gfCNCPoint4[18037] = {X 357.4015, Y 26.8104, Z -5.5000, A 0.000, B 0.000, C 0.000 }
gfCNCPoint4[18038] = {X 357.5143, Y 25.0808, Z -5.5000, A 0.000, B 0.000, C 0.000 }
gfCNCPoint4[18039] = {X 357.4620, Y 23.3484, Z -5.5000, A 0.000, B 0.000, C 0.000 }
gfCNCPoint4[18040] = {X 357.2450, Y 21.6288, Z -5.5000, A 0.000, B 0.000, C 0.000 }
gfCNCPoint4[18041] = {X 356.8838, Y 20.0827, Z -5.5000, A 0.000, B 0.000, C 0.000 }
gfCNCPoint4[18042] = {X 356.3231, Y 18.5973, Z -5.5000, A 0.000, B 0.000, C 0.000 }
gfCNCPoint4[18043] = {X 355.5723, Y 17.1983, Z -5.5000, A 0.000, B 0.000, C 0.000 }
gfCNCPoint4[18044] = {X 354.6445, Y 15.9099, Z -5.5000, A 0.000, B 0.000, C 0.000 }
gfCNCPoint4[18045] = {X 353.7511, Y 14.9589, Z -5.5000, A 0.000, B 0.000, C 0.000 }
gfCNCPoint4[18046] = {X 352.7344, Y 14.1410, Z -5.5000, A 0.000, B 0.000, C 0.000 }
gfCNCPoint4[18047] = {X 351.6142, Y 13.4719, Z -5.5000, A 0.000, B 0.000, C 0.000 }
gfCNCPoint4[18048] = {X 350.4121, Y 12.9645, Z -5.5000, A 0.000, B 0.000, C 0.000 }
gfCNCPoint4[18049] = {X 349.1512, Y 12.6287, Z -5.5000, A 0.000, B 0.000, C 0.000 }
gfCNCPoint4[18050] = {X 347.5974, Y 12.4216, Z -5.5000, A 0.000, B 0.000, C 0.000 }
gfCNCPoint4[18051] = {X 346.0300, Y 12.3943, Z -5.5000, A 0.000, B 0.000, C 0.000 }
gfCNCPoint4[18052] = {X 344.4699, Y 12.5474, Z -5.5000, A 0.000, B 0.000, C 0.000 }
gfCNCPoint4[18053] = {X 342.9377, Y 12.8786, Z -5.5000, A 0.000, B 0.000, C 0.000 }
gfCNCPoint4[18054] = {X 341.4538, Y 13.3837, Z -5.5000, A 0.000, B 0.000, C 0.000 }
gfCNCPoint4[18055] = {X 340.0376, Y 14.0559, Z -5.5000, A 0.000, B 0.000, C 0.000 }
gfCNCPoint4[18056] = {X 338.7081, Y 14.8864, Z -5.5000, A 0.000, B 0.000, C 0.000 }
gfCNCPoint4[18057] = {X 338.6941, Y 15.7112, Z -5.5000, A 0.000, B 0.000, C 0.000 }
gfCNCPoint4[18058] = {X 338.5145, Y 16.5162, Z -5.5000, A 0.000, B 0.000, C 0.000 }
gfCNCPoint4[18059] = {X 338.1767, Y 17.2687, Z -5.5000, A 0.000, B 0.000, C 0.000 }
gfCNCPoint4[18060] = {X 337.6944, Y 17.9378, Z -5.5000, A 0.000, B 0.000, C 0.000 }
gfCNCPoint4[18061] = {X 337.0874, Y 18.4963, Z -5.5000, A 0.000, B 0.000, C 0.000 }
gfCNCPoint4[18062] = {X 336.3744, Y 19.0211, Z -5.5000, A 0.000, B 0.000, C 0.000 }
gfCNCPoint4[18063] = {X 335.6039, Y 19.4547, Z -5.5000, A 0.000, B 0.000, C 0.000 }
gfCNCPoint4[18064] = {X 334.7580, Y 19.7122, Z -5.5000, A 0.000, B 0.000, C 0.000 }
gfCNCPoint4[18065] = {X 333.8766, Y 19.7814, Z -5.5000, A 0.000, B 0.000, C 0.000 }
gfCNCPoint4[18066] = {X 333.0010, Y 19.6592, Z -5.5000, A 0.000, B 0.000, C 0.000 }
gfCNCPoint4[18067] = {X 332.1722, Y 19.3511, Z -5.5000, A 0.000, B 0.000, C 0.000 }
gfCNCPoint4[18068] = {X 331.4293, Y 18.8718, Z -5.5000, A 0.000, B 0.000, C 0.000 }
gfCNCPoint4[18069] = {X 330.8071, Y 18.2436, Z -5.5000, A 0.000, B 0.000, C 0.000 }
gfCNCPoint4[18070] = {X 330.3348, Y 17.4962, Z -5.5000, A 0.000, B 0.000, C 0.000 }
gfCNCPoint4[18071] = {X 326.8100, Y 10.2453, Z -5.5000, A 0.000, B 0.000, C 0.000 }
gfCNCPoint4[18072] = {X 326.4937, Y 9.3334, Z -5.5000, A 0.000, B 0.000, C 0.000 }
gfCNCPoint4[18073] = {X 326.4004, Y 8.3728, Z -5.5000, A 0.000, B 0.000, C 0.000 }
gfCNCPoint4[18074] = {X 326.5354, Y 7.4171, Z -5.5000, A 0.000, B 0.000, C 0.000 }
gfCNCPoint4[18075] = {X 326.8911, Y 6.5199, Z -5.5000, A 0.000, B 0.000, C 0.000 }
gfCNCPoint4[18076] = {X 327.4476, Y 5.7314, Z -5.5000, A 0.000, B 0.000, C 0.000 }
gfCNCPoint4[18077] = {X 328.1737, Y 5.0956, Z -5.5000, A 0.000, B 0.000, C 0.000 }
gfCNCPoint4[18078] = {X 328.8432, Y 4.6371, Z -5.5000, A 0.000, B 0.000, C 0.000 }
gfCNCPoint4[18079] = {X 329.7003, Y 4.1969, Z -5.5000, A 0.000, B 0.000, C 0.000 }
gfCNCPoint4[18080] = {X 330.6368, Y 3.9700, Z -5.5000, A 0.000, B 0.000, C 0.000 }
gfCNCPoint4[18081] = {X 331.6003, Y 3.9690, Z -5.5000, A 0.000, B 0.000, C 0.000 }
gfCNCPoint4[18082] = {X 332.5372, Y 4.1940, Z -5.5000, A 0.000, B 0.000, C 0.000 }
gfCNCPoint4[18083] = {X 334.0587, Y 3.3390, Z -5.5000, A 0.000, B 0.000, C 0.000 }
gfCNCPoint4[18084] = {X 335.6304, Y 2.5800, Z -5.5000, A 0.000, B 0.000, C 0.000 }
gfCNCPoint4[18085] = {X 337.7472, Y 1.7211, Z -5.5000, A 0.000, B 0.000, C 0.000 }
gfCNCPoint4[18086] = {X 339.9311, Y 1.0511, Z -5.5000, A 0.000, B 0.000, C 0.000 }
gfCNCPoint4[18087] = {X 342.1653, Y 0.5751, Z -5.5000, A 0.000, B 0.000, C 0.000 }
gfCNCPoint4[18088] = {X 344.4327, Y 0.2967, Z -5.5000, A 0.000, B 0.000, C 0.000 }
gfCNCPoint4[18089] = {X 346.7157, Y 0.2181, Z -5.5000, A 0.000, B 0.000, C 0.000 }
gfCNCPoint4[18090] = {X 348.9968, Y 0.3399, Z -5.5000, A 0.000, B 0.000, C 0.000 }
gfCNCPoint4[18091] = {X 351.2585, Y 0.6611, Z -5.5000, A 0.000, B 0.000, C 0.000 }
gfCNCPoint4[18092] = {X 351.5424, Y 0.7141, Z -5.5000, A 0.000, B 0.000, C 0.000 }
gfCNCPoint4[18093] = {X 352.2774, Y -3.2178, Z -5.5000, A 0.000, B 0.000, C 0.000 }
gfCNCPoint4[18094] = {X 351.5277, Y 0.7928, Z -5.5000, A 0.000, B 0.000, C 0.000 }
gfCNCPoint4[18095] = {X 351.8094, Y 0.8454, Z -5.5000, A 0.000, B 0.000, C 0.000 }
gfCNCPoint4[18096] = {X 353.7299, Y 1.3286, Z -5.5000, A 0.000, B 0.000, C 0.000 }
gfCNCPoint4[18097] = {X 355.5955, Y 1.9932, Z -5.5000, A 0.000, B 0.000, C 0.000 }
gfCNCPoint4[18098] = {X 357.3889, Y 2.8330, Z -5.5000, A 0.000, B 0.000, C 0.000 }
gfCNCPoint4[18099] = {X 359.0939, Y 3.8404, Z -5.5000, A 0.000, B 0.000, C 0.000 }
gfCNCPoint4[18100] = {X 360.6949, Y 5.0061, Z -5.5000, A 0.000, B 0.000, C 0.000 }
gfCNCPoint4[18101] = {X 362.1770, Y 6.3196, Z -5.5000, A 0.000, B 0.000, C 0.000 }
gfCNCPoint4[18102] = {X 363.5269, Y 7.7686, Z -5.5000, A 0.000, B 0.000, C 0.000 }
gfCNCPoint4[18103] = {X 364.8608, Y 9.5026, Z -5.5000, A 0.000, B 0.000, C 0.000 }
gfCNCPoint4[18104] = {X 366.0366, Y 11.3475, Z -5.5000, A 0.000, B 0.000, C 0.000 }
gfCNCPoint4[18105] = {X 367.0451, Y 13.2890, Z -5.5000, A 0.000, B 0.000, C 0.000 }
gfCNCPoint4[18106] = {X 367.8785, Y 15.3118, Z -5.5000, A 0.000, B 0.000, C 0.000 }
gfCNCPoint4[18107] = {X 368.5301, Y 17.4002, Z -5.5000, A 0.000, B 0.000, C 0.000 }
gfCNCPoint4[18108] = {X 368.9951, Y 19.5380, Z -5.5000, A 0.000, B 0.000, C 0.000 }
gfCNCPoint4[18109] = {X 369.3083, Y 21.7425, Z -5.5000, A 0.000, B 0.000, C 0.000 }
gfCNCPoint4[18110] = {X 369.4645, Y 23.9636, Z -5.5000, A 0.000, B 0.000, C 0.000 }
gfCNCPoint4[18111] = {X 369.4630, Y 26.1902, Z -5.5000, A 0.000, B 0.000, C 0.000 }
gfCNCPoint4[18112] = {X 369.3038, Y 28.4111, Z -5.5000, A 0.000, B 0.000, C 0.000 }
gfCNCPoint4[18113] = {X 368.9876, Y 30.6151, Z -5.5000, A 0.000, B 0.000, C 0.000 }
gfCNCPoint4[18114] = {X 368.4931, Y 32.8423, Z -5.5000, A 0.000, B 0.000, C 0.000 }
gfCNCPoint4[18115] = {X 367.7916, Y 35.0132, Z -5.5000, A 0.000, B 0.000, C 0.000 }
gfCNCPoint4[18116] = {X 366.8894, Y 37.1086, Z -5.5000, A 0.000, B 0.000, C 0.000 }
gfCNCPoint4[18117] = {X 365.7944, Y 39.1101, Z -5.5000, A 0.000, B 0.000, C 0.000 }
gfCNCPoint4[18118] = {X 364.5162, Y 40.9999, Z -5.5000, A 0.000, B 0.000, C 0.000 }
gfCNCPoint4[18119] = {X 364.4010, Y 41.1577, Z -5.5000, A 0.000, B 0.000, C 0.000 }
gfCNCPoint4[18120] = {X 363.1253, Y 42.6968, Z -5.5000, A 0.000, B 0.000, C 0.000 }
gfCNCPoint4[18121] = {X 361.7132, Y 44.1118, Z -5.5000, A 0.000, B 0.000, C 0.000 }
gfCNCPoint4[18122] = {X 360.1767, Y 45.3906, Z -5.5000, A 0.000, B 0.000, C 0.000 }
gfCNCPoint4[18123] = {X 358.5288, Y 46.5223, Z -5.5000, A 0.000, B 0.000, C 0.000 }
gfCNCPoint4[18124] = {X 356.7837, Y 47.4974, Z -5.5000, A 0.000, B 0.000, C 0.000 }
gfCNCPoint4[18125] = {X 356.0912, Y 47.8253, Z -5.5000, A 0.000, B 0.000, C 0.000 }
gfCNCPoint4[18126] = {X 353.9238, Y 48.6338, Z -5.5000, A 0.000, B 0.000, C 0.000 }
gfCNCPoint4[18127] = {X 351.6854, Y 49.2177, Z -5.5000, A 0.000, B 0.000, C 0.000 }
gfCNCPoint4[18128] = {X 349.3992, Y 49.5707, Z -5.5000, A 0.000, B 0.000, C 0.000 }
gfCNCPoint4[18129] = {X 347.0889, Y 49.6893, Z -5.5000, A 0.000, B 0.000, C 0.000 }
gfCNCPoint4[18130] = {X 345.0499, Y 49.6552, Z -5.5000, A 0.000, B 0.000, C 0.000 }
gfCNCPoint4[18131] = {X 343.0216, Y 49.4445, Z -5.5000, A 0.000, B 0.000, C 0.000 }
gfCNCPoint4[18132] = {X 341.0191, Y 49.0585, Z -5.5000, A 0.000, B 0.000, C 0.000 }
gfCNCPoint4[18133] = {X 339.0577, Y 48.5004, Z -5.5000, A 0.000, B 0.000, C 0.000 }
gfCNCPoint4[18134] = {X 337.1521, Y 47.7742, Z -5.5000, A 0.000, B 0.000, C 0.000 }
gfCNCPoint4[18135] = {X 335.3167, Y 46.8855, Z -5.5000, A 0.000, B 0.000, C 0.000 }
gfCNCPoint4[18136] = {X 333.7134, Y 45.8937, Z -5.5000, A 0.000, B 0.000, C 0.000 }
gfCNCPoint4[18137] = {X 332.1949, Y 44.7763, Z -5.5000, A 0.000, B 0.000, C 0.000 }
gfCNCPoint4[18138] = {X 330.7711, Y 43.5406, Z -5.5000, A 0.000, B 0.000, C 0.000 }
gfCNCPoint4[18139] = {X 329.8559, Y 43.5681, Z -5.5000, A 0.000, B 0.000, C 0.000 }
gfCNCPoint4[18140] = {X 328.9583, Y 43.3867, Z -5.5000, A 0.000, B 0.000, C 0.000 }
gfCNCPoint4[18141] = {X 328.1256, Y 43.0059, Z -5.5000, A 0.000, B 0.000, C 0.000 }
gfCNCPoint4[18142] = {X 327.4013, Y 42.4458, Z -5.5000, A 0.000, B 0.000, C 0.000 }
gfCNCPoint4[18143] = {X 326.8042, Y 41.8634, Z -5.5000, A 0.000, B 0.000, C 0.000 }
gfCNCPoint4[18144] = {X 326.2223, Y 41.1472, Z -5.5000, A 0.000, B 0.000, C 0.000 }
gfCNCPoint4[18145] = {X 325.8201, Y 40.3166, Z -5.5000, A 0.000, B 0.000, C 0.000 }
gfCNCPoint4[18146] = {X 325.6189, Y 39.4160, Z -5.5000, A 0.000, B 0.000, C 0.000 }
gfCNCPoint4[18147] = {X 325.6294, Y 38.4932, Z -5.5000, A 0.000, B 0.000, C 0.000 }
gfCNCPoint4[18148] = {X 325.8511, Y 37.5974, Z -5.5000, A 0.000, B 0.000, C 0.000 }
gfCNCPoint4[18149] = {X 326.2722, Y 36.7763, Z -5.5000, A 0.000, B 0.000, C 0.000 }
gfCNCPoint4[18150] = {X 330.5290, Y 30.4119, Z -5.5000, A 0.000, B 0.000, C 0.000 }
gfCNCPoint4[18151] = {X 331.0932, Y 29.7536, Z -5.5000, A 0.000, B 0.000, C 0.000 }
gfCNCPoint4[18152] = {X 331.7861, Y 29.2322, Z -5.5000, A 0.000, B 0.000, C 0.000 }
gfCNCPoint4[18153] = {X 332.5750, Y 28.8724, Z -5.5000, A 0.000, B 0.000, C 0.000 }
gfCNCPoint4[18154] = {X 333.4229, Y 28.6911, Z -5.5000, A 0.000, B 0.000, C 0.000 }
gfCNCPoint4[18155] = {X 334.2900, Y 28.6968, Z -5.5000, A 0.000, B 0.000, C 0.000 }
gfCNCPoint4[18156] = {X 335.1355, Y 28.8892, Z -5.5000, A 0.000, B 0.000, C 0.000 }
gfCNCPoint4[18157] = {X 335.9196, Y 29.2593, Z -5.5000, A 0.000, B 0.000, C 0.000 }
gfCNCPoint4[18158] = {X 336.6056, Y 29.7897, Z -5.5000, A 0.000, B 0.000, C 0.000 }
gfCNCPoint4[18159] = {X 337.2041, Y 30.3665, Z -5.5000, A 0.000, B 0.000, C 0.000 }
gfCNCPoint4[18160] = {X 337.7083, Y 30.9703, Z -5.5000, A 0.000, B 0.000, C 0.000 }
gfCNCPoint4[18161] = {X 338.0846, Y 31.6611, Z -5.5000, A 0.000, B 0.000, C 0.000 }
gfCNCPoint4[18162] = {X 338.3184, Y 32.4122, Z -5.5000, A 0.000, B 0.000, C 0.000 }
gfCNCPoint4[18163] = {X 338.4007, Y 33.1945, Z -5.5000, A 0.000, B 0.000, C 0.000 }
gfCNCPoint4[18164] = {X 338.3283, Y 33.9779, Z -5.5000, A 0.000, B 0.000, C 0.000 }
gfCNCPoint4[18165] = {X 339.1660, Y 34.7396, Z -5.5000, A 0.000, B 0.000, C 0.000 }
gfCNCPoint4[18166] = {X 340.0385, Y 35.4613, Z -5.5000, A 0.000, B 0.000, C 0.000 }
gfCNCPoint4[18167] = {X 341.2965, Y 36.2941, Z -5.5000, A 0.000, B 0.000, C 0.000 }
gfCNCPoint4[18168] = {X 342.6571, Y 36.9460, Z -5.5000, A 0.000, B 0.000, C 0.000 }
gfCNCPoint4[18169] = {X 344.0944, Y 37.4045, Z -5.5000, A 0.000, B 0.000, C 0.000 }
gfCNCPoint4[18170] = {X 345.5811, Y 37.6609, Z -5.5000, A 0.000, B 0.000, C 0.000 }
gfCNCPoint4[18171] = {X 347.0889, Y 37.7104, Z -5.5000, A 0.000, B 0.000, C 0.000 }
gfCNCPoint4[18172] = {X 347.5350, Y 37.6873, Z -5.5000, A 0.000, B 0.000, C 0.000 }
gfCNCPoint4[18173] = {X 348.7314, Y 37.5466, Z -5.5000, A 0.000, B 0.000, C 0.000 }
gfCNCPoint4[18174] = {X 349.8993, Y 37.2509, Z -5.5000, A 0.000, B 0.000, C 0.000 }
gfCNCPoint4[18175] = {X 351.0187, Y 36.8054, Z -5.5000, A 0.000, B 0.000, C 0.000 }
gfCNCPoint4[18176] = {X 352.0703, Y 36.2177, Z -5.5000, A 0.000, B 0.000, C 0.000 }
gfCNCPoint4[18177] = {X 353.0363, Y 35.4978, Z -5.5000, A 0.000, B 0.000, C 0.000 }
gfCNCPoint4[18178] = {X 354.2198, Y 34.3479, Z -5.5000, A 0.000, B 0.000, C 0.000 }
gfCNCPoint4[18179] = {X 355.2441, Y 33.0542, Z -5.5000, A 0.000, B 0.000, C 0.000 }
gfCNCPoint4[18180] = {X 356.0916, Y 31.6383, Z -5.5000, A 0.000, B 0.000, C 0.000 }
gfCNCPoint4[18181] = {X 356.7482, Y 30.1245, Z -5.5000, A 0.000, B 0.000, C 0.000 }
gfCNCPoint4[18182] = {X 357.2027, Y 28.5381, Z -5.5000, A 0.000, B 0.000, C 0.000 }
gfCNCPoint4[18183] = {X 357.4809, Y 26.8196, Z -5.5000, A 0.000, B 0.000, C 0.000 }
gfCNCPoint4[18184] = {X 357.5943, Y 25.0823, Z -5.5000, A 0.000, B 0.000, C 0.000 }
gfCNCPoint4[18185] = {X 357.5418, Y 23.3422, Z -5.5000, A 0.000, B 0.000, C 0.000 }
gfCNCPoint4[18186] = {X 357.3238, Y 21.6150, Z -5.5000, A 0.000, B 0.000, C 0.000 }
gfCNCPoint4[18187] = {X 356.9602, Y 20.0588, Z -5.5000, A 0.000, B 0.000, C 0.000 }
gfCNCPoint4[18188] = {X 356.3957, Y 18.5638, Z -5.5000, A 0.000, B 0.000, C 0.000 }
gfCNCPoint4[18189] = {X 355.6400, Y 17.1558, Z -5.5000, A 0.000, B 0.000, C 0.000 }
gfCNCPoint4[18190] = {X 354.7062, Y 15.8590, Z -5.5000, A 0.000, B 0.000, C 0.000 }
gfCNCPoint4[18191] = {X 353.8052, Y 14.9000, Z -5.5000, A 0.000, B 0.000, C 0.000 }
gfCNCPoint4[18192] = {X 352.7799, Y 14.0752, Z -5.5000, A 0.000, B 0.000, C 0.000 }
gfCNCPoint4[18193] = {X 351.6502, Y 13.4005, Z -5.5000, A 0.000, B 0.000, C 0.000 }
gfCNCPoint4[18194] = {X 350.4379, Y 12.8888, Z -5.5000, A 0.000, B 0.000, C 0.000 }
gfCNCPoint4[18195] = {X 349.1664, Y 12.5502, Z -5.5000, A 0.000, B 0.000, C 0.000 }
gfCNCPoint4[18196] = {X 347.3712, Y 12.3264, Z -5.5000, A 0.000, B 0.000, C 0.000 }
gfCNCPoint4[18197] = {X 345.5623, Y 12.3410, Z -5.5000, A 0.000, B 0.000, C 0.000 }
gfCNCPoint4[18198] = {X 343.7710, Y 12.5938, Z -5.5000, A 0.000, B 0.000, C 0.000 }
gfCNCPoint4[18199] = {X 342.0287, Y 13.0804, Z -5.5000, A 0.000, B 0.000, C 0.000 }
gfCNCPoint4[18200] = {X 340.3656, Y 13.7924, Z -5.5000, A 0.000, B 0.000, C 0.000 }
gfCNCPoint4[18201] = {X 338.8108, Y 14.7172, Z -5.5000, A 0.000, B 0.000, C 0.000 }
gfCNCPoint4[18202] = {X 338.7180, Y 14.7817, Z -5.5000, A 0.000, B 0.000, C 0.000 }
gfCNCPoint4[18203] = {X 338.6257, Y 14.8469, Z -5.5000, A 0.000, B 0.000, C 0.000 }
gfCNCPoint4[18204] = {X 338.6379, Y 15.0635, Z -5.5000, A 0.000, B 0.000, C 0.000 }
gfCNCPoint4[18205] = {X 338.5596, Y 16.0358, Z -5.5000, A 0.000, B 0.000, C 0.000 }
gfCNCPoint4[18206] = {X 338.2482, Y 16.9602, Z -5.5000, A 0.000, B 0.000, C 0.000 }
gfCNCPoint4[18207] = {X 337.7223, Y 17.7818, Z -5.5000, A 0.000, B 0.000, C 0.000 }
gfCNCPoint4[18208] = {X 337.0132, Y 18.4517, Z -5.5000, A 0.000, B 0.000, C 0.000 }
gfCNCPoint4[18209] = {X 336.3278, Y 18.9560, Z -5.5000, A 0.000, B 0.000, C 0.000 }
gfCNCPoint4[18210] = {X 335.5713, Y 19.3817, Z -5.5000, A 0.000, B 0.000, C 0.000 }
gfCNCPoint4[18211] = {X 334.7407, Y 19.6341, Z -5.5000, A 0.000, B 0.000, C 0.000 }
gfCNCPoint4[18212] = {X 333.8753, Y 19.7014, Z -5.5000, A 0.000, B 0.000, C 0.000 }
gfCNCPoint4[18213] = {X 333.0157, Y 19.5804, Z -5.5000, A 0.000, B 0.000, C 0.000 }
gfCNCPoint4[18214] = {X 332.2025, Y 19.2768, Z -5.5000, A 0.000, B 0.000, C 0.000 }
gfCNCPoint4[18215] = {X 331.4739, Y 18.8049, Z -5.5000, A 0.000, B 0.000, C 0.000 }
gfCNCPoint4[18216] = {X 330.8643, Y 18.1870, Z -5.5000, A 0.000, B 0.000, C 0.000 }
gfCNCPoint4[18217] = {X 330.4023, Y 17.4521, Z -5.5000, A 0.000, B 0.000, C 0.000 }
gfCNCPoint4[18218] = {X 326.8820, Y 10.2103, Z -5.5000, A 0.000, B 0.000, C 0.000 }
gfCNCPoint4[18219] = {X 326.5719, Y 9.3163, Z -5.5000, A 0.000, B 0.000, C 0.000 }
gfCNCPoint4[18220] = {X 326.4804, Y 8.3746, Z -5.5000, A 0.000, B 0.000, C 0.000 }
gfCNCPoint4[18221] = {X 326.6127, Y 7.4376, Z -5.5000, A 0.000, B 0.000, C 0.000 }
gfCNCPoint4[18222] = {X 326.9614, Y 6.5580, Z -5.5000, A 0.000, B 0.000, C 0.000 }
gfCNCPoint4[18223] = {X 327.5070, Y 5.7849, Z -5.5000, A 0.000, B 0.000, C 0.000 }
gfCNCPoint4[18224] = {X 328.2189, Y 5.1616, Z -5.5000, A 0.000, B 0.000, C 0.000 }
gfCNCPoint4[18225] = {X 328.8880, Y 4.7034, Z -5.5000, A 0.000, B 0.000, C 0.000 }
gfCNCPoint4[18226] = {X 329.7043, Y 4.2813, Z -5.5000, A 0.000, B 0.000, C 0.000 }
gfCNCPoint4[18227] = {X 330.5954, Y 4.0567, Z -5.5000, A 0.000, B 0.000, C 0.000 }
gfCNCPoint4[18228] = {X 331.5142, Y 4.0413, Z -5.5000, A 0.000, B 0.000, C 0.000 }
gfCNCPoint4[18229] = {X 332.4122, Y 4.2361, Z -5.5000, A 0.000, B 0.000, C 0.000 }
gfCNCPoint4[18230] = {X 332.5467, Y 4.2817, Z -5.5000, A 0.000, B 0.000, C 0.000 }
gfCNCPoint4[18231] = {X 332.6255, Y 4.2342, Z -5.5000, A 0.000, B 0.000, C 0.000 }
gfCNCPoint4[18232] = {X 332.7044, Y 4.1870, Z -5.5000, A 0.000, B 0.000, C 0.000 }
gfCNCPoint4[18233] = {X 334.1609, Y 3.3760, Z -5.5000, A 0.000, B 0.000, C 0.000 }
gfCNCPoint4[18234] = {X 335.6629, Y 2.6530, Z -5.5000, A 0.000, B 0.000, C 0.000 }
gfCNCPoint4[18235] = {X 336.0092, Y 2.4989, Z -5.5000, A 0.000, B 0.000, C 0.000 }
gfCNCPoint4[18236] = {X 338.0805, Y 1.6908, Z -5.5000, A 0.000, B 0.000, C 0.000 }
gfCNCPoint4[18237] = {X 340.2133, Y 1.0629, Z -5.5000, A 0.000, B 0.000, C 0.000 }
gfCNCPoint4[18238] = {X 342.3920, Y 0.6199, Z -5.5000, A 0.000, B 0.000, C 0.000 }
gfCNCPoint4[18239] = {X 344.6007, Y 0.3648, Z -5.5000, A 0.000, B 0.000, C 0.000 }
gfCNCPoint4[18240] = {X 346.8231, Y 0.2997, Z -5.5000, A 0.000, B 0.000, C 0.000 }
gfCNCPoint4[18241] = {X 349.0429, Y 0.4250, Z -5.5000, A 0.000, B 0.000, C 0.000 }
gfCNCPoint4[18242] = {X 351.2438, Y 0.7397, Z -5.5000, A 0.000, B 0.000, C 0.000 }
gfCNCPoint4[18243] = {X 351.5277, Y 0.7928, Z -5.5000, A 0.000, B 0.000, C 0.000 }
gfCNCPoint4[18244] = {X 352.2774, Y -3.2178, Z -5.5000, A 0.000, B 0.000, C 0.000 }
gfCNCPoint4[18245] = {X 352.2774, Y -3.2178, Z -2.5000, A 0.000, B 0.000, C 0.000 }
gfCNCPoint4[18246] = {X 352.2774, Y -3.2178, Z 11.0000, A 0.000, B 0.000, C 0.000 }
gfCNCPoint4[18247] = {X 606.0427, Y 42.9006, Z 11.0000, A 0.000, B 0.000, C 0.000 }
gfCNCPoint4[18248] = {X 606.0427, Y 42.9006, Z -2.5000, A 0.000, B 0.000, C 0.000 }
gfCNCPoint4[18249] = {X 606.0427, Y 42.9006, Z -5.5000, A 0.000, B 0.000, C 0.000 }
gfCNCPoint4[18250] = {X 603.6966, Y 47.0767, Z -5.5000, A 0.000, B 0.000, C 0.000 }
gfCNCPoint4[18251] = {X 603.6311, Y 47.1892, Z -5.5000, A 0.000, B 0.000, C 0.000 }
gfCNCPoint4[18252] = {X 603.5622, Y 47.2997, Z -5.5000, A 0.000, B 0.000, C 0.000 }
gfCNCPoint4[18253] = {X 603.0358, Y 47.9600, Z -5.5000, A 0.000, B 0.000, C 0.000 }
gfCNCPoint4[18254] = {X 602.3889, Y 48.5030, Z -5.5000, A 0.000, B 0.000, C 0.000 }
gfCNCPoint4[18255] = {X 601.6473, Y 48.9069, Z -5.5000, A 0.000, B 0.000, C 0.000 }
gfCNCPoint4[18256] = {X 600.8403, Y 49.1559, Z -5.5000, A 0.000, B 0.000, C 0.000 }
gfCNCPoint4[18257] = {X 600.0000, Y 49.2400, Z -5.5000, A 0.000, B 0.000, C 0.000 }
gfCNCPoint4[18258] = {X 593.5565, Y 49.2400, Z -5.5000, A 0.000, B 0.000, C 0.000 }
gfCNCPoint4[18259] = {X 592.6130, Y 49.1337, Z -5.5000, A 0.000, B 0.000, C 0.000 }
gfCNCPoint4[18260] = {X 591.7169, Y 48.8201, Z -5.5000, A 0.000, B 0.000, C 0.000 }
gfCNCPoint4[18261] = {X 590.9129, Y 48.3150, Z -5.5000, A 0.000, B 0.000, C 0.000 }
gfCNCPoint4[18262] = {X 590.2416, Y 47.6436, Z -5.5000, A 0.000, B 0.000, C 0.000 }
gfCNCPoint4[18263] = {X 589.7364, Y 46.8397, Z -5.5000, A 0.000, B 0.000, C 0.000 }
gfCNCPoint4[18264] = {X 589.4228, Y 45.9435, Z -5.5000, A 0.000, B 0.000, C 0.000 }
gfCNCPoint4[18265] = {X 589.3165, Y 45.0000, Z -5.5000, A 0.000, B 0.000, C 0.000 }
gfCNCPoint4[18266] = {X 589.3165, Y 44.0650, Z -5.5000, A 0.000, B 0.000, C 0.000 }
gfCNCPoint4[18267] = {X 589.4207, Y 43.1447, Z -5.5000, A 0.000, B 0.000, C 0.000 }
gfCNCPoint4[18268] = {X 589.7204, Y 42.2685, Z -5.5000, A 0.000, B 0.000, C 0.000 }
gfCNCPoint4[18269] = {X 590.2017, Y 41.4773, Z -5.5000, A 0.000, B 0.000, C 0.000 }
gfCNCPoint4[18270] = {X 590.8419, Y 40.8081, Z -5.5000, A 0.000, B 0.000, C 0.000 }
gfCNCPoint4[18271] = {X 590.8425, Y 33.1211, Z -5.5000, A 0.000, B 0.000, C 0.000 }
gfCNCPoint4[18272] = {X 585.3714, Y 46.6218, Z -5.5000, A 0.000, B 0.000, C 0.000 }
gfCNCPoint4[18273] = {X 585.0085, Y 47.3114, Z -5.5000, A 0.000, B 0.000, C 0.000 }
gfCNCPoint4[18274] = {X 584.5255, Y 47.9228, Z -5.5000, A 0.000, B 0.000, C 0.000 }
gfCNCPoint4[18275] = {X 583.9387, Y 48.4356, Z -5.5000, A 0.000, B 0.000, C 0.000 }
gfCNCPoint4[18276] = {X 583.2680, Y 48.8323, Z -5.5000, A 0.000, B 0.000, C 0.000 }
gfCNCPoint4[18277] = {X 582.3418, Y 49.1460, Z -5.5000, A 0.000, B 0.000, C 0.000 }
gfCNCPoint4[18278] = {X 581.3682, Y 49.2391, Z -5.5000, A 0.000, B 0.000, C 0.000 }
gfCNCPoint4[18279] = {X 580.3993, Y 49.1068, Z -5.5000, A 0.000, B 0.000, C 0.000 }
gfCNCPoint4[18280] = {X 579.4864, Y 48.7559, Z -5.5000, A 0.000, B 0.000, C 0.000 }
gfCNCPoint4[18281] = {X 578.6782, Y 48.2052, Z -5.5000, A 0.000, B 0.000, C 0.000 }
gfCNCPoint4[18282] = {X 578.0177, Y 47.4840, Z -5.5000, A 0.000, B 0.000, C 0.000 }
gfCNCPoint4[18283] = {X 577.5400, Y 46.6307, Z -5.5000, A 0.000, B 0.000, C 0.000 }
gfCNCPoint4[18284] = {X 571.9392, Y 32.9353, Z -5.5000, A 0.000, B 0.000, C 0.000 }
gfCNCPoint4[18285] = {X 571.9395, Y 40.8083, Z -5.5000, A 0.000, B 0.000, C 0.000 }
gfCNCPoint4[18286] = {X 571.9710, Y 40.8341, Z -5.5000, A 0.000, B 0.000, C 0.000 }
gfCNCPoint4[18287] = {X 572.5961, Y 41.4925, Z -5.5000, A 0.000, B 0.000, C 0.000 }
gfCNCPoint4[18288] = {X 573.0668, Y 42.2689, Z -5.5000, A 0.000, B 0.000, C 0.000 }
gfCNCPoint4[18289] = {X 573.3613, Y 43.1276, Z -5.5000, A 0.000, B 0.000, C 0.000 }
gfCNCPoint4[18290] = {X 573.4663, Y 44.0294, Z -5.5000, A 0.000, B 0.000, C 0.000 }
gfCNCPoint4[18291] = {X 573.4664, Y 45.0000, Z -5.5000, A 0.000, B 0.000, C 0.000 }
gfCNCPoint4[18292] = {X 573.3601, Y 45.9435, Z -5.5000, A 0.000, B 0.000, C 0.000 }
gfCNCPoint4[18293] = {X 573.0465, Y 46.8397, Z -5.5000, A 0.000, B 0.000, C 0.000 }
gfCNCPoint4[18294] = {X 572.5414, Y 47.6436, Z -5.5000, A 0.000, B 0.000, C 0.000 }
gfCNCPoint4[18295] = {X 571.8700, Y 48.3150, Z -5.5000, A 0.000, B 0.000, C 0.000 }
gfCNCPoint4[18296] = {X 571.0661, Y 48.8201, Z -5.5000, A 0.000, B 0.000, C 0.000 }
gfCNCPoint4[18297] = {X 570.1699, Y 49.1337, Z -5.5000, A 0.000, B 0.000, C 0.000 }
gfCNCPoint4[18298] = {X 569.2264, Y 49.2400, Z -5.5000, A 0.000, B 0.000, C 0.000 }
gfCNCPoint4[18299] = {X 562.4443, Y 49.2400, Z -5.5000, A 0.000, B 0.000, C 0.000 }
gfCNCPoint4[18300] = {X 561.5008, Y 49.1337, Z -5.5000, A 0.000, B 0.000, C 0.000 }
gfCNCPoint4[18301] = {X 560.6046, Y 48.8201, Z -5.5000, A 0.000, B 0.000, C 0.000 }
gfCNCPoint4[18302] = {X 559.8007, Y 48.3150, Z -5.5000, A 0.000, B 0.000, C 0.000 }
gfCNCPoint4[18303] = {X 559.1293, Y 47.6436, Z -5.5000, A 0.000, B 0.000, C 0.000 }
gfCNCPoint4[18304] = {X 558.6242, Y 46.8397, Z -5.5000, A 0.000, B 0.000, C 0.000 }
gfCNCPoint4[18305] = {X 558.3106, Y 45.9435, Z -5.5000, A 0.000, B 0.000, C 0.000 }
gfCNCPoint4[18306] = {X 558.2043, Y 45.0000, Z -5.5000, A 0.000, B 0.000, C 0.000 }
gfCNCPoint4[18307] = {X 558.2043, Y 44.0651, Z -5.5000, A 0.000, B 0.000, C 0.000 }
gfCNCPoint4[18308] = {X 558.3083, Y 43.1444, Z -5.5000, A 0.000, B 0.000, C 0.000 }
gfCNCPoint4[18309] = {X 558.6083, Y 42.2679, Z -5.5000, A 0.000, B 0.000, C 0.000 }
gfCNCPoint4[18310] = {X 559.0903, Y 41.4766, Z -5.5000, A 0.000, B 0.000, C 0.000 }
gfCNCPoint4[18311] = {X 559.7315, Y 40.8078, Z -5.5000, A 0.000, B 0.000, C 0.000 }
gfCNCPoint4[18312] = {X 559.7315, Y 9.1926, Z -5.5000, A 0.000, B 0.000, C 0.000 }
gfCNCPoint4[18313] = {X 559.0937, Y 8.5323, Z -5.5000, A 0.000, B 0.000, C 0.000 }
gfCNCPoint4[18314] = {X 558.6129, Y 7.7502, Z -5.5000, A 0.000, B 0.000, C 0.000 }
gfCNCPoint4[18315] = {X 558.3118, Y 6.8829, Z -5.5000, A 0.000, B 0.000, C 0.000 }
gfCNCPoint4[18316] = {X 558.2045, Y 5.9711, Z -5.5000, A 0.000, B 0.000, C 0.000 }
gfCNCPoint4[18317] = {X 558.2043, Y 5.0000, Z -5.5000, A 0.000, B 0.000, C 0.000 }
gfCNCPoint4[18318] = {X 558.3106, Y 4.0565, Z -5.5000, A 0.000, B 0.000, C 0.000 }
gfCNCPoint4[18319] = {X 558.6242, Y 3.1603, Z -5.5000, A 0.000, B 0.000, C 0.000 }
gfCNCPoint4[18320] = {X 559.1293, Y 2.3564, Z -5.5000, A 0.000, B 0.000, C 0.000 }
gfCNCPoint4[18321] = {X 559.8007, Y 1.6850, Z -5.5000, A 0.000, B 0.000, C 0.000 }
gfCNCPoint4[18322] = {X 560.6046, Y 1.1799, Z -5.5000, A 0.000, B 0.000, C 0.000 }
gfCNCPoint4[18323] = {X 561.5008, Y 0.8663, Z -5.5000, A 0.000, B 0.000, C 0.000 }
gfCNCPoint4[18324] = {X 562.4443, Y 0.7600, Z -5.5000, A 0.000, B 0.000, C 0.000 }
gfCNCPoint4[18325] = {X 570.9376, Y 0.7600, Z -5.5000, A 0.000, B 0.000, C 0.000 }
gfCNCPoint4[18326] = {X 571.8810, Y 0.8663, Z -5.5000, A 0.000, B 0.000, C 0.000 }
gfCNCPoint4[18327] = {X 572.7772, Y 1.1799, Z -5.5000, A 0.000, B 0.000, C 0.000 }
gfCNCPoint4[18328] = {X 573.5812, Y 1.6850, Z -5.5000, A 0.000, B 0.000, C 0.000 }
gfCNCPoint4[18329] = {X 574.2525, Y 2.3564, Z -5.5000, A 0.000, B 0.000, C 0.000 }
gfCNCPoint4[18330] = {X 574.7577, Y 3.1603, Z -5.5000, A 0.000, B 0.000, C 0.000 }
gfCNCPoint4[18331] = {X 575.0712, Y 4.0565, Z -5.5000, A 0.000, B 0.000, C 0.000 }
gfCNCPoint4[18332] = {X 575.1776, Y 5.0000, Z -5.5000, A 0.000, B 0.000, C 0.000 }
gfCNCPoint4[18333] = {X 575.1776, Y 5.9342, Z -5.5000, A 0.000, B 0.000, C 0.000 }
gfCNCPoint4[18334] = {X 575.1024, Y 6.7290, Z -5.5000, A 0.000, B 0.000, C 0.000 }
gfCNCPoint4[18335] = {X 574.8796, Y 7.4955, Z -5.5000, A 0.000, B 0.000, C 0.000 }
gfCNCPoint4[18336] = {X 574.5170, Y 8.2067, Z -5.5000, A 0.000, B 0.000, C 0.000 }
gfCNCPoint4[18337] = {X 581.1908, Y 24.5812, Z -5.5000, A 0.000, B 0.000, C 0.000 }
gfCNCPoint4[18338] = {X 587.9347, Y 8.0878, Z -5.5000, A 0.000, B 0.000, C 0.000 }
gfCNCPoint4[18339] = {X 587.6158, Y 7.4198, Z -5.5000, A 0.000, B 0.000, C 0.000 }
gfCNCPoint4[18340] = {X 587.4179, Y 6.7066, Z -5.5000, A 0.000, B 0.000, C 0.000 }
gfCNCPoint4[18341] = {X 587.3471, Y 5.9698, Z -5.5000, A 0.000, B 0.000, C 0.000 }
gfCNCPoint4[18342] = {X 587.3470, Y 5.0000, Z -5.5000, A 0.000, B 0.000, C 0.000 }
gfCNCPoint4[18343] = {X 587.4533, Y 4.0565, Z -5.5000, A 0.000, B 0.000, C 0.000 }
gfCNCPoint4[18344] = {X 587.7668, Y 3.1603, Z -5.5000, A 0.000, B 0.000, C 0.000 }
gfCNCPoint4[18345] = {X 588.2720, Y 2.3564, Z -5.5000, A 0.000, B 0.000, C 0.000 }
gfCNCPoint4[18346] = {X 588.9434, Y 1.6850, Z -5.5000, A 0.000, B 0.000, C 0.000 }
gfCNCPoint4[18347] = {X 589.7473, Y 1.1799, Z -5.5000, A 0.000, B 0.000, C 0.000 }
gfCNCPoint4[18348] = {X 590.6435, Y 0.8663, Z -5.5000, A 0.000, B 0.000, C 0.000 }
gfCNCPoint4[18349] = {X 591.5870, Y 0.7600, Z -5.5000, A 0.000, B 0.000, C 0.000 }
gfCNCPoint4[18350] = {X 600.0000, Y 0.7600, Z -5.5000, A 0.000, B 0.000, C 0.000 }
gfCNCPoint4[18351] = {X 600.8403, Y 0.8441, Z -5.5000, A 0.000, B 0.000, C 0.000 }
gfCNCPoint4[18352] = {X 601.6473, Y 1.0931, Z -5.5000, A 0.000, B 0.000, C 0.000 }
gfCNCPoint4[18353] = {X 602.3889, Y 1.4970, Z -5.5000, A 0.000, B 0.000, C 0.000 }
gfCNCPoint4[18354] = {X 603.0358, Y 2.0400, Z -5.5000, A 0.000, B 0.000, C 0.000 }
gfCNCPoint4[18355] = {X 603.5622, Y 2.7003, Z -5.5000, A 0.000, B 0.000, C 0.000 }
gfCNCPoint4[18356] = {X 603.6311, Y 2.8108, Z -5.5000, A 0.000, B 0.000, C 0.000 }
gfCNCPoint4[18357] = {X 603.6966, Y 2.9233, Z -5.5000, A 0.000, B 0.000, C 0.000 }
gfCNCPoint4[18358] = {X 607.8228, Y 10.2681, Z -5.5000, A 0.000, B 0.000, C 0.000 }
gfCNCPoint4[18359] = {X 607.8228, Y 10.2681, Z -2.5000, A 0.000, B 0.000, C 0.000 }
gfCNCPoint4[18360] = {X 607.8228, Y 10.2681, Z 11.0000, A 0.000, B 0.000, C 0.000 }
gfCNCPoint4[18361] = {X 607.6966, Y 39.1586, Z 11.0000, A 0.000, B 0.000, C 0.000 }
gfCNCPoint4[18362] = {X 607.6966, Y 39.1586, Z -2.5000, A 0.000, B 0.000, C 0.000 }
gfCNCPoint4[18363] = {X 607.6966, Y 39.1586, Z -5.5000, A 0.000, B 0.000, C 0.000 }
gfCNCPoint4[18364] = {X 603.6966, Y 46.9081, Z -5.5000, A 0.000, B 0.000, C 0.000 }
gfCNCPoint4[18365] = {X 603.6000, Y 47.0846, Z -5.5000, A 0.000, B 0.000, C 0.000 }
gfCNCPoint4[18366] = {X 603.4950, Y 47.2563, Z -5.5000, A 0.000, B 0.000, C 0.000 }
gfCNCPoint4[18367] = {X 602.9785, Y 47.9042, Z -5.5000, A 0.000, B 0.000, C 0.000 }
gfCNCPoint4[18368] = {X 602.3438, Y 48.4369, Z -5.5000, A 0.000, B 0.000, C 0.000 }
gfCNCPoint4[18369] = {X 601.6162, Y 48.8332, Z -5.5000, A 0.000, B 0.000, C 0.000 }
gfCNCPoint4[18370] = {X 600.8245, Y 49.0775, Z -5.5000, A 0.000, B 0.000, C 0.000 }
gfCNCPoint4[18371] = {X 600.0000, Y 49.1600, Z -5.5000, A 0.000, B 0.000, C 0.000 }
gfCNCPoint4[18372] = {X 593.5565, Y 49.1600, Z -5.5000, A 0.000, B 0.000, C 0.000 }
gfCNCPoint4[18373] = {X 592.6308, Y 49.0557, Z -5.5000, A 0.000, B 0.000, C 0.000 }
gfCNCPoint4[18374] = {X 591.7516, Y 48.7480, Z -5.5000, A 0.000, B 0.000, C 0.000 }
gfCNCPoint4[18375] = {X 590.9628, Y 48.2524, Z -5.5000, A 0.000, B 0.000, C 0.000 }
gfCNCPoint4[18376] = {X 590.3041, Y 47.5937, Z -5.5000, A 0.000, B 0.000, C 0.000 }
gfCNCPoint4[18377] = {X 589.8085, Y 46.8050, Z -5.5000, A 0.000, B 0.000, C 0.000 }
gfCNCPoint4[18378] = {X 589.5008, Y 45.9257, Z -5.5000, A 0.000, B 0.000, C 0.000 }
gfCNCPoint4[18379] = {X 589.3965, Y 45.0000, Z -5.5000, A 0.000, B 0.000, C 0.000 }
gfCNCPoint4[18380] = {X 589.3965, Y 44.0653, Z -5.5000, A 0.000, B 0.000, C 0.000 }
gfCNCPoint4[18381] = {X 589.5008, Y 43.1532, Z -5.5000, A 0.000, B 0.000, C 0.000 }
gfCNCPoint4[18382] = {X 589.8008, Y 42.2856, Z -5.5000, A 0.000, B 0.000, C 0.000 }
gfCNCPoint4[18383] = {X 590.2822, Y 41.5040, Z -5.5000, A 0.000, B 0.000, C 0.000 }
gfCNCPoint4[18384] = {X 590.9219, Y 40.8456, Z -5.5000, A 0.000, B 0.000, C 0.000 }
gfCNCPoint4[18385] = {X 590.9226, Y 32.7106, Z -5.5000, A 0.000, B 0.000, C 0.000 }
gfCNCPoint4[18386] = {X 585.2975, Y 46.5912, Z -5.5000, A 0.000, B 0.000, C 0.000 }
gfCNCPoint4[18387] = {X 584.9414, Y 47.2678, Z -5.5000, A 0.000, B 0.000, C 0.000 }
gfCNCPoint4[18388] = {X 584.4675, Y 47.8677, Z -5.5000, A 0.000, B 0.000, C 0.000 }
gfCNCPoint4[18389] = {X 583.8918, Y 48.3708, Z -5.5000, A 0.000, B 0.000, C 0.000 }
gfCNCPoint4[18390] = {X 583.2338, Y 48.7600, Z -5.5000, A 0.000, B 0.000, C 0.000 }
gfCNCPoint4[18391] = {X 582.3250, Y 49.0678, Z -5.5000, A 0.000, B 0.000, C 0.000 }
gfCNCPoint4[18392] = {X 581.3699, Y 49.1592, Z -5.5000, A 0.000, B 0.000, C 0.000 }
gfCNCPoint4[18393] = {X 580.4192, Y 49.0293, Z -5.5000, A 0.000, B 0.000, C 0.000 }
gfCNCPoint4[18394] = {X 579.5236, Y 48.6850, Z -5.5000, A 0.000, B 0.000, C 0.000 }
gfCNCPoint4[18395] = {X 578.7306, Y 48.1448, Z -5.5000, A 0.000, B 0.000, C 0.000 }
gfCNCPoint4[18396] = {X 578.0826, Y 47.4372, Z -5.5000, A 0.000, B 0.000, C 0.000 }
gfCNCPoint4[18397] = {X 577.6138, Y 46.5999, Z -5.5000, A 0.000, B 0.000, C 0.000 }
gfCNCPoint4[18398] = {X 571.8592, Y 32.5283, Z -5.5000, A 0.000, B 0.000, C 0.000 }
gfCNCPoint4[18399] = {X 571.8595, Y 40.8462, Z -5.5000, A 0.000, B 0.000, C 0.000 }
gfCNCPoint4[18400] = {X 571.9198, Y 40.8955, Z -5.5000, A 0.000, B 0.000, C 0.000 }
gfCNCPoint4[18401] = {X 572.5329, Y 41.5415, Z -5.5000, A 0.000, B 0.000, C 0.000 }
gfCNCPoint4[18402] = {X 572.9944, Y 42.3031, Z -5.5000, A 0.000, B 0.000, C 0.000 }
gfCNCPoint4[18403] = {X 573.2833, Y 43.1455, Z -5.5000, A 0.000, B 0.000, C 0.000 }
gfCNCPoint4[18404] = {X 573.3863, Y 44.0301, Z -5.5000, A 0.000, B 0.000, C 0.000 }
gfCNCPoint4[18405] = {X 573.3864, Y 45.0000, Z -5.5000, A 0.000, B 0.000, C 0.000 }
gfCNCPoint4[18406] = {X 573.2821, Y 45.9257, Z -5.5000, A 0.000, B 0.000, C 0.000 }
gfCNCPoint4[18407] = {X 572.9745, Y 46.8050, Z -5.5000, A 0.000, B 0.000, C 0.000 }
gfCNCPoint4[18408] = {X 572.4788, Y 47.5937, Z -5.5000, A 0.000, B 0.000, C 0.000 }
gfCNCPoint4[18409] = {X 571.8201, Y 48.2524, Z -5.5000, A 0.000, B 0.000, C 0.000 }
gfCNCPoint4[18410] = {X 571.0314, Y 48.7480, Z -5.5000, A 0.000, B 0.000, C 0.000 }
gfCNCPoint4[18411] = {X 570.1521, Y 49.0557, Z -5.5000, A 0.000, B 0.000, C 0.000 }
gfCNCPoint4[18412] = {X 569.2264, Y 49.1600, Z -5.5000, A 0.000, B 0.000, C 0.000 }
gfCNCPoint4[18413] = {X 562.4443, Y 49.1600, Z -5.5000, A 0.000, B 0.000, C 0.000 }
gfCNCPoint4[18414] = {X 561.5186, Y 49.0557, Z -5.5000, A 0.000, B 0.000, C 0.000 }
gfCNCPoint4[18415] = {X 560.6393, Y 48.7480, Z -5.5000, A 0.000, B 0.000, C 0.000 }
gfCNCPoint4[18416] = {X 559.8506, Y 48.2524, Z -5.5000, A 0.000, B 0.000, C 0.000 }
gfCNCPoint4[18417] = {X 559.1919, Y 47.5937, Z -5.5000, A 0.000, B 0.000, C 0.000 }
gfCNCPoint4[18418] = {X 558.6963, Y 46.8050, Z -5.5000, A 0.000, B 0.000, C 0.000 }
gfCNCPoint4[18419] = {X 558.3886, Y 45.9257, Z -5.5000, A 0.000, B 0.000, C 0.000 }
gfCNCPoint4[18420] = {X 558.2843, Y 45.0000, Z -5.5000, A 0.000, B 0.000, C 0.000 }
gfCNCPoint4[18421] = {X 558.2843, Y 44.0654, Z -5.5000, A 0.000, B 0.000, C 0.000 }
gfCNCPoint4[18422] = {X 558.3884, Y 43.1529, Z -5.5000, A 0.000, B 0.000, C 0.000 }
gfCNCPoint4[18423] = {X 558.6887, Y 42.2850, Z -5.5000, A 0.000, B 0.000, C 0.000 }
gfCNCPoint4[18424] = {X 559.1708, Y 41.5033, Z -5.5000, A 0.000, B 0.000, C 0.000 }
gfCNCPoint4[18425] = {X 559.8115, Y 40.8454, Z -5.5000, A 0.000, B 0.000, C 0.000 }
gfCNCPoint4[18426] = {X 559.8115, Y 9.1549, Z -5.5000, A 0.000, B 0.000, C 0.000 }
gfCNCPoint4[18427] = {X 559.1741, Y 8.5054, Z -5.5000, A 0.000, B 0.000, C 0.000 }
gfCNCPoint4[18428] = {X 558.6933, Y 7.7328, Z -5.5000, A 0.000, B 0.000, C 0.000 }
gfCNCPoint4[18429] = {X 558.3919, Y 6.8741, Z -5.5000, A 0.000, B 0.000, C 0.000 }
gfCNCPoint4[18430] = {X 558.2845, Y 5.9704, Z -5.5000, A 0.000, B 0.000, C 0.000 }
gfCNCPoint4[18431] = {X 558.2843, Y 5.0000, Z -5.5000, A 0.000, B 0.000, C 0.000 }
gfCNCPoint4[18432] = {X 558.3886, Y 4.0743, Z -5.5000, A 0.000, B 0.000, C 0.000 }
gfCNCPoint4[18433] = {X 558.6963, Y 3.1950, Z -5.5000, A 0.000, B 0.000, C 0.000 }
gfCNCPoint4[18434] = {X 559.1919, Y 2.4063, Z -5.5000, A 0.000, B 0.000, C 0.000 }
gfCNCPoint4[18435] = {X 559.8506, Y 1.7476, Z -5.5000, A 0.000, B 0.000, C 0.000 }
gfCNCPoint4[18436] = {X 560.6393, Y 1.2520, Z -5.5000, A 0.000, B 0.000, C 0.000 }
gfCNCPoint4[18437] = {X 561.5186, Y 0.9443, Z -5.5000, A 0.000, B 0.000, C 0.000 }
gfCNCPoint4[18438] = {X 562.4443, Y 0.8400, Z -5.5000, A 0.000, B 0.000, C 0.000 }
gfCNCPoint4[18439] = {X 570.9376, Y 0.8400, Z -5.5000, A 0.000, B 0.000, C 0.000 }
gfCNCPoint4[18440] = {X 571.8632, Y 0.9443, Z -5.5000, A 0.000, B 0.000, C 0.000 }
gfCNCPoint4[18441] = {X 572.7425, Y 1.2520, Z -5.5000, A 0.000, B 0.000, C 0.000 }
gfCNCPoint4[18442] = {X 573.5313, Y 1.7476, Z -5.5000, A 0.000, B 0.000, C 0.000 }
gfCNCPoint4[18443] = {X 574.1900, Y 2.4063, Z -5.5000, A 0.000, B 0.000, C 0.000 }
gfCNCPoint4[18444] = {X 574.6856, Y 3.1950, Z -5.5000, A 0.000, B 0.000, C 0.000 }
gfCNCPoint4[18445] = {X 574.9933, Y 4.0743, Z -5.5000, A 0.000, B 0.000, C 0.000 }
gfCNCPoint4[18446] = {X 575.0976, Y 5.0000, Z -5.5000, A 0.000, B 0.000, C 0.000 }
gfCNCPoint4[18447] = {X 575.0976, Y 5.9342, Z -5.5000, A 0.000, B 0.000, C 0.000 }
gfCNCPoint4[18448] = {X 575.0212, Y 6.7274, Z -5.5000, A 0.000, B 0.000, C 0.000 }
gfCNCPoint4[18449] = {X 574.7950, Y 7.4915, Z -5.5000, A 0.000, B 0.000, C 0.000 }
gfCNCPoint4[18450] = {X 574.4273, Y 8.1985, Z -5.5000, A 0.000, B 0.000, C 0.000 }
gfCNCPoint4[18451] = {X 581.1907, Y 24.7928, Z -5.5000, A 0.000, B 0.000, C 0.000 }
gfCNCPoint4[18452] = {X 588.0238, Y 8.0811, Z -5.5000, A 0.000, B 0.000, C 0.000 }
gfCNCPoint4[18453] = {X 587.7000, Y 7.4164, Z -5.5000, A 0.000, B 0.000, C 0.000 }
gfCNCPoint4[18454] = {X 587.4990, Y 6.7050, Z -5.5000, A 0.000, B 0.000, C 0.000 }
gfCNCPoint4[18455] = {X 587.4271, Y 5.9692, Z -5.5000, A 0.000, B 0.000, C 0.000 }
gfCNCPoint4[18456] = {X 587.4270, Y 5.0000, Z -5.5000, A 0.000, B 0.000, C 0.000 }
gfCNCPoint4[18457] = {X 587.5313, Y 4.0743, Z -5.5000, A 0.000, B 0.000, C 0.000 }
gfCNCPoint4[18458] = {X 587.8389, Y 3.1950, Z -5.5000, A 0.000, B 0.000, C 0.000 }
gfCNCPoint4[18459] = {X 588.3345, Y 2.4063, Z -5.5000, A 0.000, B 0.000, C 0.000 }
gfCNCPoint4[18460] = {X 588.9932, Y 1.7476, Z -5.5000, A 0.000, B 0.000, C 0.000 }
gfCNCPoint4[18461] = {X 589.7820, Y 1.2520, Z -5.5000, A 0.000, B 0.000, C 0.000 }
gfCNCPoint4[18462] = {X 590.6613, Y 0.9443, Z -5.5000, A 0.000, B 0.000, C 0.000 }
gfCNCPoint4[18463] = {X 591.5870, Y 0.8400, Z -5.5000, A 0.000, B 0.000, C 0.000 }
gfCNCPoint4[18464] = {X 600.0000, Y 0.8400, Z -5.5000, A 0.000, B 0.000, C 0.000 }
gfCNCPoint4[18465] = {X 600.8245, Y 0.9225, Z -5.5000, A 0.000, B 0.000, C 0.000 }
gfCNCPoint4[18466] = {X 601.6162, Y 1.1668, Z -5.5000, A 0.000, B 0.000, C 0.000 }
gfCNCPoint4[18467] = {X 602.3438, Y 1.5631, Z -5.5000, A 0.000, B 0.000, C 0.000 }
gfCNCPoint4[18468] = {X 602.9785, Y 2.0958, Z -5.5000, A 0.000, B 0.000, C 0.000 }
gfCNCPoint4[18469] = {X 603.4950, Y 2.7437, Z -5.5000, A 0.000, B 0.000, C 0.000 }
gfCNCPoint4[18470] = {X 603.6000, Y 2.9154, Z -5.5000, A 0.000, B 0.000, C 0.000 }
gfCNCPoint4[18471] = {X 603.6966, Y 3.0919, Z -5.5000, A 0.000, B 0.000, C 0.000 }
gfCNCPoint4[18472] = {X 607.6966, Y 10.8414, Z -5.5000, A 0.000, B 0.000, C 0.000 }
gfCNCPoint4[18473] = {X 607.6966, Y 10.8414, Z -2.5000, A 0.000, B 0.000, C 0.000 }
gfCNCPoint4[18474] = {X 607.6966, Y 10.8414, Z 11.0000, A 0.000, B 0.000, C 0.000 }
gfCNCPoint4[18475] = {X 607.6966, Y 38.1633, Z 11.0000, A 0.000, B 0.000, C 0.000 }
gfCNCPoint4[18476] = {X 607.6966, Y 38.1633, Z -2.5000, A 0.000, B 0.000, C 0.000 }
gfCNCPoint4[18477] = {X 607.6966, Y 38.1633, Z -5.5000, A 0.000, B 0.000, C 0.000 }
gfCNCPoint4[18478] = {X 603.6966, Y 46.7267, Z -5.5000, A 0.000, B 0.000, C 0.000 }
gfCNCPoint4[18479] = {X 603.5705, Y 46.9744, Z -5.5000, A 0.000, B 0.000, C 0.000 }
gfCNCPoint4[18480] = {X 603.4278, Y 47.2129, Z -5.5000, A 0.000, B 0.000, C 0.000 }
gfCNCPoint4[18481] = {X 602.9212, Y 47.8483, Z -5.5000, A 0.000, B 0.000, C 0.000 }
gfCNCPoint4[18482] = {X 602.2988, Y 48.3708, Z -5.5000, A 0.000, B 0.000, C 0.000 }
gfCNCPoint4[18483] = {X 601.5851, Y 48.7595, Z -5.5000, A 0.000, B 0.000, C 0.000 }
gfCNCPoint4[18484] = {X 600.8086, Y 48.9991, Z -5.5000, A 0.000, B 0.000, C 0.000 }
gfCNCPoint4[18485] = {X 600.0000, Y 49.0800, Z -5.5000, A 0.000, B 0.000, C 0.000 }
gfCNCPoint4[18486] = {X 593.5565, Y 49.0800, Z -5.5000, A 0.000, B 0.000, C 0.000 }
gfCNCPoint4[18487] = {X 592.6486, Y 48.9777, Z -5.5000, A 0.000, B 0.000, C 0.000 }
gfCNCPoint4[18488] = {X 591.7863, Y 48.6760, Z -5.5000, A 0.000, B 0.000, C 0.000 }
gfCNCPoint4[18489] = {X 591.0127, Y 48.1899, Z -5.5000, A 0.000, B 0.000, C 0.000 }
gfCNCPoint4[18490] = {X 590.3667, Y 47.5438, Z -5.5000, A 0.000, B 0.000, C 0.000 }
gfCNCPoint4[18491] = {X 589.8806, Y 46.7702, Z -5.5000, A 0.000, B 0.000, C 0.000 }
gfCNCPoint4[18492] = {X 589.5788, Y 45.9079, Z -5.5000, A 0.000, B 0.000, C 0.000 }
gfCNCPoint4[18493] = {X 589.4765, Y 45.0000, Z -5.5000, A 0.000, B 0.000, C 0.000 }
gfCNCPoint4[18494] = {X 589.4765, Y 44.0656, Z -5.5000, A 0.000, B 0.000, C 0.000 }
gfCNCPoint4[18495] = {X 589.5731, Y 43.1967, Z -5.5000, A 0.000, B 0.000, C 0.000 }
gfCNCPoint4[18496] = {X 589.8508, Y 42.3677, Z -5.5000, A 0.000, B 0.000, C 0.000 }
gfCNCPoint4[18497] = {X 590.2973, Y 41.6160, Z -5.5000, A 0.000, B 0.000, C 0.000 }
gfCNCPoint4[18498] = {X 590.8924, Y 40.9754, Z -5.5000, A 0.000, B 0.000, C 0.000 }
gfCNCPoint4[18499] = {X 590.9467, Y 40.9290, Z -5.5000, A 0.000, B 0.000, C 0.000 }
gfCNCPoint4[18500] = {X 591.0019, Y 40.8835, Z -5.5000, A 0.000, B 0.000, C 0.000 }
gfCNCPoint4[18501] = {X 591.0026, Y 32.3001, Z -5.5000, A 0.000, B 0.000, C 0.000 }
gfCNCPoint4[18502] = {X 585.2236, Y 46.5606, Z -5.5000, A 0.000, B 0.000, C 0.000 }
gfCNCPoint4[18503] = {X 584.8743, Y 47.2242, Z -5.5000, A 0.000, B 0.000, C 0.000 }
gfCNCPoint4[18504] = {X 584.4095, Y 47.8125, Z -5.5000, A 0.000, B 0.000, C 0.000 }
gfCNCPoint4[18505] = {X 583.8449, Y 48.3059, Z -5.5000, A 0.000, B 0.000, C 0.000 }
gfCNCPoint4[18506] = {X 583.1996, Y 48.6877, Z -5.5000, A 0.000, B 0.000, C 0.000 }
gfCNCPoint4[18507] = {X 582.3082, Y 48.9895, Z -5.5000, A 0.000, B 0.000, C 0.000 }
gfCNCPoint4[18508] = {X 581.3715, Y 49.0792, Z -5.5000, A 0.000, B 0.000, C 0.000 }
gfCNCPoint4[18509] = {X 580.4391, Y 48.9518, Z -5.5000, A 0.000, B 0.000, C 0.000 }
gfCNCPoint4[18510] = {X 579.5607, Y 48.6142, Z -5.5000, A 0.000, B 0.000, C 0.000 }
gfCNCPoint4[18511] = {X 578.7830, Y 48.0843, Z -5.5000, A 0.000, B 0.000, C 0.000 }
gfCNCPoint4[18512] = {X 578.1474, Y 47.3903, Z -5.5000, A 0.000, B 0.000, C 0.000 }
gfCNCPoint4[18513] = {X 577.6877, Y 46.5692, Z -5.5000, A 0.000, B 0.000, C 0.000 }
gfCNCPoint4[18514] = {X 571.7792, Y 32.1213, Z -5.5000, A 0.000, B 0.000, C 0.000 }
gfCNCPoint4[18515] = {X 571.7795, Y 40.8841, Z -5.5000, A 0.000, B 0.000, C 0.000 }
gfCNCPoint4[18516] = {X 571.8685, Y 40.9570, Z -5.5000, A 0.000, B 0.000, C 0.000 }
gfCNCPoint4[18517] = {X 572.4696, Y 41.5904, Z -5.5000, A 0.000, B 0.000, C 0.000 }
gfCNCPoint4[18518] = {X 572.9221, Y 42.3373, Z -5.5000, A 0.000, B 0.000, C 0.000 }
gfCNCPoint4[18519] = {X 573.2053, Y 43.1634, Z -5.5000, A 0.000, B 0.000, C 0.000 }
gfCNCPoint4[18520] = {X 573.3063, Y 44.0308, Z -5.5000, A 0.000, B 0.000, C 0.000 }
gfCNCPoint4[18521] = {X 573.3064, Y 45.0000, Z -5.5000, A 0.000, B 0.000, C 0.000 }
gfCNCPoint4[18522] = {X 573.2041, Y 45.9079, Z -5.5000, A 0.000, B 0.000, C 0.000 }
gfCNCPoint4[18523] = {X 572.9024, Y 46.7702, Z -5.5000, A 0.000, B 0.000, C 0.000 }
gfCNCPoint4[18524] = {X 572.4163, Y 47.5438, Z -5.5000, A 0.000, B 0.000, C 0.000 }
gfCNCPoint4[18525] = {X 571.7703, Y 48.1899, Z -5.5000, A 0.000, B 0.000, C 0.000 }
gfCNCPoint4[18526] = {X 570.9967, Y 48.6760, Z -5.5000, A 0.000, B 0.000, C 0.000 }
gfCNCPoint4[18527] = {X 570.1343, Y 48.9777, Z -5.5000, A 0.000, B 0.000, C 0.000 }
gfCNCPoint4[18528] = {X 569.2264, Y 49.0800, Z -5.5000, A 0.000, B 0.000, C 0.000 }
gfCNCPoint4[18529] = {X 562.4443, Y 49.0800, Z -5.5000, A 0.000, B 0.000, C 0.000 }
gfCNCPoint4[18530] = {X 561.5364, Y 48.9777, Z -5.5000, A 0.000, B 0.000, C 0.000 }
gfCNCPoint4[18531] = {X 560.6741, Y 48.6760, Z -5.5000, A 0.000, B 0.000, C 0.000 }
gfCNCPoint4[18532] = {X 559.9005, Y 48.1899, Z -5.5000, A 0.000, B 0.000, C 0.000 }
gfCNCPoint4[18533] = {X 559.2544, Y 47.5438, Z -5.5000, A 0.000, B 0.000, C 0.000 }
gfCNCPoint4[18534] = {X 558.7683, Y 46.7702, Z -5.5000, A 0.000, B 0.000, C 0.000 }
gfCNCPoint4[18535] = {X 558.4666, Y 45.9079, Z -5.5000, A 0.000, B 0.000, C 0.000 }
gfCNCPoint4[18536] = {X 558.3643, Y 45.0000, Z -5.5000, A 0.000, B 0.000, C 0.000 }
gfCNCPoint4[18537] = {X 558.3643, Y 44.0657, Z -5.5000, A 0.000, B 0.000, C 0.000 }
gfCNCPoint4[18538] = {X 558.4685, Y 43.1615, Z -5.5000, A 0.000, B 0.000, C 0.000 }
gfCNCPoint4[18539] = {X 558.7691, Y 42.3023, Z -5.5000, A 0.000, B 0.000, C 0.000 }
gfCNCPoint4[18540] = {X 559.2513, Y 41.5304, Z -5.5000, A 0.000, B 0.000, C 0.000 }
gfCNCPoint4[18541] = {X 559.8915, Y 40.8834, Z -5.5000, A 0.000, B 0.000, C 0.000 }
gfCNCPoint4[18542] = {X 559.8915, Y 9.1167, Z -5.5000, A 0.000, B 0.000, C 0.000 }
gfCNCPoint4[18543] = {X 559.8355, Y 9.0711, Z -5.5000, A 0.000, B 0.000, C 0.000 }
gfCNCPoint4[18544] = {X 559.7804, Y 9.0244, Z -5.5000, A 0.000, B 0.000, C 0.000 }
gfCNCPoint4[18545] = {X 559.1882, Y 8.3925, Z -5.5000, A 0.000, B 0.000, C 0.000 }
gfCNCPoint4[18546] = {X 558.7426, Y 7.6499, Z -5.5000, A 0.000, B 0.000, C 0.000 }
gfCNCPoint4[18547] = {X 558.4639, Y 6.8300, Z -5.5000, A 0.000, B 0.000, C 0.000 }
gfCNCPoint4[18548] = {X 558.3645, Y 5.9697, Z -5.5000, A 0.000, B 0.000, C 0.000 }
gfCNCPoint4[18549] = {X 558.3643, Y 5.0000, Z -5.5000, A 0.000, B 0.000, C 0.000 }
gfCNCPoint4[18550] = {X 558.4666, Y 4.0921, Z -5.5000, A 0.000, B 0.000, C 0.000 }
gfCNCPoint4[18551] = {X 558.7683, Y 3.2298, Z -5.5000, A 0.000, B 0.000, C 0.000 }
gfCNCPoint4[18552] = {X 559.2544, Y 2.4562, Z -5.5000, A 0.000, B 0.000, C 0.000 }
gfCNCPoint4[18553] = {X 559.9005, Y 1.8101, Z -5.5000, A 0.000, B 0.000, C 0.000 }
gfCNCPoint4[18554] = {X 560.6741, Y 1.3240, Z -5.5000, A 0.000, B 0.000, C 0.000 }
gfCNCPoint4[18555] = {X 561.5364, Y 1.0223, Z -5.5000, A 0.000, B 0.000, C 0.000 }
gfCNCPoint4[18556] = {X 562.4443, Y 0.9200, Z -5.5000, A 0.000, B 0.000, C 0.000 }
gfCNCPoint4[18557] = {X 570.9376, Y 0.9200, Z -5.5000, A 0.000, B 0.000, C 0.000 }
gfCNCPoint4[18558] = {X 571.8454, Y 1.0223, Z -5.5000, A 0.000, B 0.000, C 0.000 }
gfCNCPoint4[18559] = {X 572.7078, Y 1.3240, Z -5.5000, A 0.000, B 0.000, C 0.000 }
gfCNCPoint4[18560] = {X 573.4814, Y 1.8101, Z -5.5000, A 0.000, B 0.000, C 0.000 }
gfCNCPoint4[18561] = {X 574.1274, Y 2.4562, Z -5.5000, A 0.000, B 0.000, C 0.000 }
gfCNCPoint4[18562] = {X 574.6135, Y 3.2298, Z -5.5000, A 0.000, B 0.000, C 0.000 }
gfCNCPoint4[18563] = {X 574.9153, Y 4.0921, Z -5.5000, A 0.000, B 0.000, C 0.000 }
gfCNCPoint4[18564] = {X 575.0176, Y 5.0000, Z -5.5000, A 0.000, B 0.000, C 0.000 }
gfCNCPoint4[18565] = {X 575.0176, Y 5.9342, Z -5.5000, A 0.000, B 0.000, C 0.000 }
gfCNCPoint4[18566] = {X 574.9500, Y 6.6735, Z -5.5000, A 0.000, B 0.000, C 0.000 }
gfCNCPoint4[18567] = {X 574.7496, Y 7.3882, Z -5.5000, A 0.000, B 0.000, C 0.000 }
gfCNCPoint4[18568] = {X 574.4231, Y 8.0548, Z -5.5000, A 0.000, B 0.000, C 0.000 }
gfCNCPoint4[18569] = {X 574.3787, Y 8.1261, Z -5.5000, A 0.000, B 0.000, C 0.000 }
gfCNCPoint4[18570] = {X 574.3328, Y 8.1965, Z -5.5000, A 0.000, B 0.000, C 0.000 }
gfCNCPoint4[18571] = {X 574.3589, Y 8.2416, Z -5.5000, A 0.000, B 0.000, C 0.000 }
gfCNCPoint4[18572] = {X 581.1906, Y 25.0045, Z -5.5000, A 0.000, B 0.000, C 0.000 }
gfCNCPoint4[18573] = {X 588.1132, Y 8.0740, Z -5.5000, A 0.000, B 0.000, C 0.000 }
gfCNCPoint4[18574] = {X 588.0737, Y 8.0085, Z -5.5000, A 0.000, B 0.000, C 0.000 }
gfCNCPoint4[18575] = {X 588.0354, Y 7.9423, Z -5.5000, A 0.000, B 0.000, C 0.000 }
gfCNCPoint4[18576] = {X 587.7486, Y 7.3174, Z -5.5000, A 0.000, B 0.000, C 0.000 }
gfCNCPoint4[18577] = {X 587.5708, Y 6.6531, Z -5.5000, A 0.000, B 0.000, C 0.000 }
gfCNCPoint4[18578] = {X 587.5071, Y 5.9685, Z -5.5000, A 0.000, B 0.000, C 0.000 }
gfCNCPoint4[18579] = {X 587.5070, Y 5.0000, Z -5.5000, A 0.000, B 0.000, C 0.000 }
gfCNCPoint4[18580] = {X 587.6092, Y 4.0921, Z -5.5000, A 0.000, B 0.000, C 0.000 }
gfCNCPoint4[18581] = {X 587.9110, Y 3.2298, Z -5.5000, A 0.000, B 0.000, C 0.000 }
gfCNCPoint4[18582] = {X 588.3971, Y 2.4562, Z -5.5000, A 0.000, B 0.000, C 0.000 }
gfCNCPoint4[18583] = {X 589.0431, Y 1.8101, Z -5.5000, A 0.000, B 0.000, C 0.000 }
gfCNCPoint4[18584] = {X 589.8167, Y 1.3240, Z -5.5000, A 0.000, B 0.000, C 0.000 }
gfCNCPoint4[18585] = {X 590.6791, Y 1.0223, Z -5.5000, A 0.000, B 0.000, C 0.000 }
gfCNCPoint4[18586] = {X 591.5870, Y 0.9200, Z -5.5000, A 0.000, B 0.000, C 0.000 }
gfCNCPoint4[18587] = {X 600.0000, Y 0.9200, Z -5.5000, A 0.000, B 0.000, C 0.000 }
gfCNCPoint4[18588] = {X 600.8086, Y 1.0009, Z -5.5000, A 0.000, B 0.000, C 0.000 }
gfCNCPoint4[18589] = {X 601.5851, Y 1.2405, Z -5.5000, A 0.000, B 0.000, C 0.000 }
gfCNCPoint4[18590] = {X 602.2988, Y 1.6292, Z -5.5000, A 0.000, B 0.000, C 0.000 }
gfCNCPoint4[18591] = {X 602.9212, Y 2.1517, Z -5.5000, A 0.000, B 0.000, C 0.000 }
gfCNCPoint4[18592] = {X 603.4278, Y 2.7871, Z -5.5000, A 0.000, B 0.000, C 0.000 }
gfCNCPoint4[18593] = {X 603.5705, Y 3.0256, Z -5.5000, A 0.000, B 0.000, C 0.000 }
gfCNCPoint4[18594] = {X 603.6966, Y 3.2733, Z -5.5000, A 0.000, B 0.000, C 0.000 }
gfCNCPoint4[18595] = {X 607.6966, Y 11.8367, Z -5.5000, A 0.000, B 0.000, C 0.000 }
gfCNCPoint4[18596] = {X 607.6966, Y 11.8367, Z -2.5000, A 0.000, B 0.000, C 0.000 }
gfCNCPoint4[18597] = {X 607.6966, Y 11.8367, Z 11.0000, A 0.000, B 0.000, C 0.000 }
gfCNCPoint4[18598] = {X 607.6966, Y 36.8518, Z 11.0000, A 0.000, B 0.000, C 0.000 }
gfCNCPoint4[18599] = {X 607.6966, Y 36.8518, Z -2.5000, A 0.000, B 0.000, C 0.000 }
gfCNCPoint4[18600] = {X 607.6966, Y 36.8518, Z -5.5000, A 0.000, B 0.000, C 0.000 }
gfCNCPoint4[18601] = {X 603.6966, Y 46.5281, Z -5.5000, A 0.000, B 0.000, C 0.000 }
gfCNCPoint4[18602] = {X 603.5431, Y 46.8564, Z -5.5000, A 0.000, B 0.000, C 0.000 }
gfCNCPoint4[18603] = {X 603.3606, Y 47.1695, Z -5.5000, A 0.000, B 0.000, C 0.000 }
gfCNCPoint4[18604] = {X 602.8639, Y 47.7925, Z -5.5000, A 0.000, B 0.000, C 0.000 }
gfCNCPoint4[18605] = {X 602.2537, Y 48.3047, Z -5.5000, A 0.000, B 0.000, C 0.000 }
gfCNCPoint4[18606] = {X 601.5540, Y 48.6858, Z -5.5000, A 0.000, B 0.000, C 0.000 }
gfCNCPoint4[18607] = {X 600.7927, Y 48.9207, Z -5.5000, A 0.000, B 0.000, C 0.000 }
gfCNCPoint4[18608] = {X 600.0000, Y 49.0000, Z -5.5000, A 0.000, B 0.000, C 0.000 }
gfCNCPoint4[18609] = {X 593.5565, Y 49.0000, Z -5.5000, A 0.000, B 0.000, C 0.000 }
gfCNCPoint4[18610] = {X 592.6664, Y 48.8997, Z -5.5000, A 0.000, B 0.000, C 0.000 }
gfCNCPoint4[18611] = {X 591.8210, Y 48.6039, Z -5.5000, A 0.000, B 0.000, C 0.000 }
gfCNCPoint4[18612] = {X 591.0626, Y 48.1273, Z -5.5000, A 0.000, B 0.000, C 0.000 }
gfCNCPoint4[18613] = {X 590.4292, Y 47.4940, Z -5.5000, A 0.000, B 0.000, C 0.000 }
gfCNCPoint4[18614] = {X 589.9527, Y 46.7355, Z -5.5000, A 0.000, B 0.000, C 0.000 }
gfCNCPoint4[18615] = {X 589.6568, Y 45.8901, Z -5.5000, A 0.000, B 0.000, C 0.000 }
gfCNCPoint4[18616] = {X 589.5565, Y 45.0000, Z -5.5000, A 0.000, B 0.000, C 0.000 }
gfCNCPoint4[18617] = {X 589.5565, Y 44.0660, Z -5.5000, A 0.000, B 0.000, C 0.000 }
gfCNCPoint4[18618] = {X 589.6512, Y 43.2139, Z -5.5000, A 0.000, B 0.000, C 0.000 }
gfCNCPoint4[18619] = {X 589.9236, Y 42.4010, Z -5.5000, A 0.000, B 0.000, C 0.000 }
gfCNCPoint4[18620] = {X 590.3614, Y 41.6639, Z -5.5000, A 0.000, B 0.000, C 0.000 }
gfCNCPoint4[18621] = {X 590.9449, Y 41.0358, Z -5.5000, A 0.000, B 0.000, C 0.000 }
gfCNCPoint4[18622] = {X 591.0127, Y 40.9781, Z -5.5000, A 0.000, B 0.000, C 0.000 }
gfCNCPoint4[18623] = {X 591.0818, Y 40.9219, Z -5.5000, A 0.000, B 0.000, C 0.000 }
gfCNCPoint4[18624] = {X 591.0838, Y 40.3075, Z -5.5000, A 0.000, B 0.000, C 0.000 }
gfCNCPoint4[18625] = {X 591.0826, Y 32.0436, Z -5.5000, A 0.000, B 0.000, C 0.000 }
gfCNCPoint4[18626] = {X 590.9675, Y 32.1736, Z -5.5000, A 0.000, B 0.000, C 0.000 }
gfCNCPoint4[18627] = {X 590.3121, Y 33.7910, Z -5.5000, A 0.000, B 0.000, C 0.000 }
gfCNCPoint4[18628] = {X 585.1497, Y 46.5300, Z -5.5000, A 0.000, B 0.000, C 0.000 }
gfCNCPoint4[18629] = {X 584.8073, Y 47.1805, Z -5.5000, A 0.000, B 0.000, C 0.000 }
gfCNCPoint4[18630] = {X 584.3516, Y 47.7574, Z -5.5000, A 0.000, B 0.000, C 0.000 }
gfCNCPoint4[18631] = {X 583.7980, Y 48.2411, Z -5.5000, A 0.000, B 0.000, C 0.000 }
gfCNCPoint4[18632] = {X 583.1653, Y 48.6154, Z -5.5000, A 0.000, B 0.000, C 0.000 }
gfCNCPoint4[18633] = {X 582.2878, Y 48.9121, Z -5.5000, A 0.000, B 0.000, C 0.000 }
gfCNCPoint4[18634] = {X 581.3656, Y 48.9990, Z -5.5000, A 0.000, B 0.000, C 0.000 }
gfCNCPoint4[18635] = {X 580.4480, Y 48.8715, Z -5.5000, A 0.000, B 0.000, C 0.000 }
gfCNCPoint4[18636] = {X 579.5845, Y 48.5363, Z -5.5000, A 0.000, B 0.000, C 0.000 }
gfCNCPoint4[18637] = {X 578.8212, Y 48.0115, Z -5.5000, A 0.000, B 0.000, C 0.000 }
gfCNCPoint4[18638] = {X 578.1990, Y 47.3251, Z -5.5000, A 0.000, B 0.000, C 0.000 }
gfCNCPoint4[18639] = {X 577.7515, Y 46.5141, Z -5.5000, A 0.000, B 0.000, C 0.000 }
gfCNCPoint4[18640] = {X 571.6992, Y 31.7143, Z -5.5000, A 0.000, B 0.000, C 0.000 }
gfCNCPoint4[18641] = {X 571.6995, Y 40.9220, Z -5.5000, A 0.000, B 0.000, C 0.000 }
gfCNCPoint4[18642] = {X 571.8383, Y 41.0364, Z -5.5000, A 0.000, B 0.000, C 0.000 }
gfCNCPoint4[18643] = {X 572.4241, Y 41.6628, Z -5.5000, A 0.000, B 0.000, C 0.000 }
gfCNCPoint4[18644] = {X 572.8629, Y 42.3998, Z -5.5000, A 0.000, B 0.000, C 0.000 }
gfCNCPoint4[18645] = {X 573.1345, Y 43.2133, Z -5.5000, A 0.000, B 0.000, C 0.000 }
gfCNCPoint4[18646] = {X 573.2264, Y 44.0660, Z -5.5000, A 0.000, B 0.000, C 0.000 }
gfCNCPoint4[18647] = {X 573.2264, Y 45.0000, Z -5.5000, A 0.000, B 0.000, C 0.000 }
gfCNCPoint4[18648] = {X 573.1261, Y 45.8901, Z -5.5000, A 0.000, B 0.000, C 0.000 }
gfCNCPoint4[18649] = {X 572.8303, Y 46.7355, Z -5.5000, A 0.000, B 0.000, C 0.000 }
gfCNCPoint4[18650] = {X 572.3538, Y 47.4940, Z -5.5000, A 0.000, B 0.000, C 0.000 }
gfCNCPoint4[18651] = {X 571.7204, Y 48.1273, Z -5.5000, A 0.000, B 0.000, C 0.000 }
gfCNCPoint4[18652] = {X 570.9620, Y 48.6039, Z -5.5000, A 0.000, B 0.000, C 0.000 }
gfCNCPoint4[18653] = {X 570.1165, Y 48.8997, Z -5.5000, A 0.000, B 0.000, C 0.000 }
gfCNCPoint4[18654] = {X 569.2264, Y 49.0000, Z -5.5000, A 0.000, B 0.000, C 0.000 }
gfCNCPoint4[18655] = {X 562.4443, Y 49.0000, Z -5.5000, A 0.000, B 0.000, C 0.000 }
gfCNCPoint4[18656] = {X 561.5542, Y 48.8997, Z -5.5000, A 0.000, B 0.000, C 0.000 }
gfCNCPoint4[18657] = {X 560.7088, Y 48.6039, Z -5.5000, A 0.000, B 0.000, C 0.000 }
gfCNCPoint4[18658] = {X 559.9503, Y 48.1273, Z -5.5000, A 0.000, B 0.000, C 0.000 }
gfCNCPoint4[18659] = {X 559.3170, Y 47.4940, Z -5.5000, A 0.000, B 0.000, C 0.000 }
gfCNCPoint4[18660] = {X 558.8404, Y 46.7355, Z -5.5000, A 0.000, B 0.000, C 0.000 }
gfCNCPoint4[18661] = {X 558.5446, Y 45.8901, Z -5.5000, A 0.000, B 0.000, C 0.000 }
gfCNCPoint4[18662] = {X 558.4443, Y 45.0000, Z -5.5000, A 0.000, B 0.000, C 0.000 }
gfCNCPoint4[18663] = {X 558.4443, Y 44.0660, Z -5.5000, A 0.000, B 0.000, C 0.000 }
gfCNCPoint4[18664] = {X 558.5486, Y 43.1701, Z -5.5000, A 0.000, B 0.000, C 0.000 }
gfCNCPoint4[18665] = {X 558.8495, Y 42.3198, Z -5.5000, A 0.000, B 0.000, C 0.000 }
gfCNCPoint4[18666] = {X 559.3318, Y 41.5577, Z -5.5000, A 0.000, B 0.000, C 0.000 }
gfCNCPoint4[18667] = {X 559.9715, Y 40.9218, Z -5.5000, A 0.000, B 0.000, C 0.000 }
gfCNCPoint4[18668] = {X 559.9715, Y 9.0781, Z -5.5000, A 0.000, B 0.000, C 0.000 }
gfCNCPoint4[18669] = {X 559.9014, Y 9.0217, Z -5.5000, A 0.000, B 0.000, C 0.000 }
gfCNCPoint4[18670] = {X 559.8326, Y 8.9638, Z -5.5000, A 0.000, B 0.000, C 0.000 }
gfCNCPoint4[18671] = {X 559.2467, Y 8.3373, Z -5.5000, A 0.000, B 0.000, C 0.000 }
gfCNCPoint4[18672] = {X 558.8079, Y 7.6004, Z -5.5000, A 0.000, B 0.000, C 0.000 }
gfCNCPoint4[18673] = {X 558.5362, Y 6.7868, Z -5.5000, A 0.000, B 0.000, C 0.000 }
gfCNCPoint4[18674] = {X 558.4443, Y 5.9340, Z -5.5000, A 0.000, B 0.000, C 0.000 }
gfCNCPoint4[18675] = {X 558.4443, Y 5.0000, Z -5.5000, A 0.000, B 0.000, C 0.000 }
gfCNCPoint4[18676] = {X 558.5446, Y 4.1099, Z -5.5000, A 0.000, B 0.000, C 0.000 }
gfCNCPoint4[18677] = {X 558.8404, Y 3.2645, Z -5.5000, A 0.000, B 0.000, C 0.000 }
gfCNCPoint4[18678] = {X 559.3170, Y 2.5060, Z -5.5000, A 0.000, B 0.000, C 0.000 }
gfCNCPoint4[18679] = {X 559.9503, Y 1.8727, Z -5.5000, A 0.000, B 0.000, C 0.000 }
gfCNCPoint4[18680] = {X 560.7088, Y 1.3961, Z -5.5000, A 0.000, B 0.000, C 0.000 }
gfCNCPoint4[18681] = {X 561.5542, Y 1.1003, Z -5.5000, A 0.000, B 0.000, C 0.000 }
gfCNCPoint4[18682] = {X 562.4443, Y 1.0000, Z -5.5000, A 0.000, B 0.000, C 0.000 }
gfCNCPoint4[18683] = {X 570.9376, Y 1.0000, Z -5.5000, A 0.000, B 0.000, C 0.000 }
gfCNCPoint4[18684] = {X 571.8276, Y 1.1003, Z -5.5000, A 0.000, B 0.000, C 0.000 }
gfCNCPoint4[18685] = {X 572.6731, Y 1.3961, Z -5.5000, A 0.000, B 0.000, C 0.000 }
gfCNCPoint4[18686] = {X 573.4315, Y 1.8727, Z -5.5000, A 0.000, B 0.000, C 0.000 }
gfCNCPoint4[18687] = {X 574.0649, Y 2.5060, Z -5.5000, A 0.000, B 0.000, C 0.000 }
gfCNCPoint4[18688] = {X 574.5414, Y 3.2645, Z -5.5000, A 0.000, B 0.000, C 0.000 }
gfCNCPoint4[18689] = {X 574.8373, Y 4.1099, Z -5.5000, A 0.000, B 0.000, C 0.000 }
gfCNCPoint4[18690] = {X 574.9376, Y 5.0000, Z -5.5000, A 0.000, B 0.000, C 0.000 }
gfCNCPoint4[18691] = {X 574.9372, Y 5.9858, Z -5.5000, A 0.000, B 0.000, C 0.000 }
gfCNCPoint4[18692] = {X 574.8649, Y 6.6927, Z -5.5000, A 0.000, B 0.000, C 0.000 }
gfCNCPoint4[18693] = {X 574.6687, Y 7.3757, Z -5.5000, A 0.000, B 0.000, C 0.000 }
gfCNCPoint4[18694] = {X 574.3547, Y 8.0132, Z -5.5000, A 0.000, B 0.000, C 0.000 }
gfCNCPoint4[18695] = {X 574.2920, Y 8.1130, Z -5.5000, A 0.000, B 0.000, C 0.000 }
gfCNCPoint4[18696] = {X 574.2264, Y 8.2108, Z -5.5000, A 0.000, B 0.000, C 0.000 }
gfCNCPoint4[18697] = {X 574.2614, Y 8.2359, Z -5.5000, A 0.000, B 0.000, C 0.000 }
gfCNCPoint4[18698] = {X 574.2849, Y 8.2721, Z -5.5000, A 0.000, B 0.000, C 0.000 }
gfCNCPoint4[18699] = {X 574.9161, Y 9.8074, Z -5.5000, A 0.000, B 0.000, C 0.000 }
gfCNCPoint4[18700] = {X 581.1904, Y 25.2163, Z -5.5000, A 0.000, B 0.000, C 0.000 }
gfCNCPoint4[18701] = {X 588.2027, Y 8.0664, Z -5.5000, A 0.000, B 0.000, C 0.000 }
gfCNCPoint4[18702] = {X 588.1529, Y 7.9852, Z -5.5000, A 0.000, B 0.000, C 0.000 }
gfCNCPoint4[18703] = {X 588.1051, Y 7.9029, Z -5.5000, A 0.000, B 0.000, C 0.000 }
gfCNCPoint4[18704] = {X 587.8201, Y 7.2796, Z -5.5000, A 0.000, B 0.000, C 0.000 }
gfCNCPoint4[18705] = {X 587.6457, Y 6.6168, Z -5.5000, A 0.000, B 0.000, C 0.000 }
gfCNCPoint4[18706] = {X 587.5870, Y 5.9340, Z -5.5000, A 0.000, B 0.000, C 0.000 }
gfCNCPoint4[18707] = {X 587.5870, Y 5.0000, Z -5.5000, A 0.000, B 0.000, C 0.000 }
gfCNCPoint4[18708] = {X 587.6872, Y 4.1099, Z -5.5000, A 0.000, B 0.000, C 0.000 }
gfCNCPoint4[18709] = {X 587.9831, Y 3.2645, Z -5.5000, A 0.000, B 0.000, C 0.000 }
gfCNCPoint4[18710] = {X 588.4596, Y 2.5060, Z -5.5000, A 0.000, B 0.000, C 0.000 }
gfCNCPoint4[18711] = {X 589.0930, Y 1.8727, Z -5.5000, A 0.000, B 0.000, C 0.000 }
gfCNCPoint4[18712] = {X 589.8514, Y 1.3961, Z -5.5000, A 0.000, B 0.000, C 0.000 }
gfCNCPoint4[18713] = {X 590.6969, Y 1.1003, Z -5.5000, A 0.000, B 0.000, C 0.000 }
gfCNCPoint4[18714] = {X 591.5870, Y 1.0000, Z -5.5000, A 0.000, B 0.000, C 0.000 }
gfCNCPoint4[18715] = {X 600.0000, Y 1.0000, Z -5.5000, A 0.000, B 0.000, C 0.000 }
gfCNCPoint4[18716] = {X 600.7927, Y 1.0793, Z -5.5000, A 0.000, B 0.000, C 0.000 }
gfCNCPoint4[18717] = {X 601.5540, Y 1.3142, Z -5.5000, A 0.000, B 0.000, C 0.000 }
gfCNCPoint4[18718] = {X 602.2537, Y 1.6953, Z -5.5000, A 0.000, B 0.000, C 0.000 }
gfCNCPoint4[18719] = {X 602.8639, Y 2.2075, Z -5.5000, A 0.000, B 0.000, C 0.000 }
gfCNCPoint4[18720] = {X 603.3606, Y 2.8305, Z -5.5000, A 0.000, B 0.000, C 0.000 }
gfCNCPoint4[18721] = {X 603.5431, Y 3.1436, Z -5.5000, A 0.000, B 0.000, C 0.000 }
gfCNCPoint4[18722] = {X 603.6966, Y 3.4719, Z -5.5000, A 0.000, B 0.000, C 0.000 }
gfCNCPoint4[18723] = {X 607.6966, Y 13.1482, Z -5.5000, A 0.000, B 0.000, C 0.000 }
gfCNCPoint4[18724] = {X 607.6966, Y 13.1482, Z -2.5000, A 0.000, B 0.000, C 0.000 }
gfCNCPoint4[18725] = {X 607.6966, Y 13.1482, Z 11.0000, A 0.000, B 0.000, C 0.000 }
gfCNCPoint4[18726] = {X 448.7141, Y 19.7821, Z 11.0000, A 0.000, B 0.000, C 0.000 }
gfCNCPoint4[18727] = {X 448.7141, Y 19.7821, Z -1.6667, A 0.000, B 0.000, C 0.000 }
gfCNCPoint4[18728] = {X 444.0414, Y 19.7821, Z -2.9187, A 0.000, B 0.000, C 0.000 }
gfCNCPoint4[18729] = {X 443.3487, Y 19.7983, Z -3.1044, A 0.000, B 0.000, C 0.000 }
gfCNCPoint4[18730] = {X 442.7490, Y 19.8051, Z -3.2651, A 0.000, B 0.000, C 0.000 }
gfCNCPoint4[18731] = {X 442.0369, Y 19.9283, Z -3.4587, A 0.000, B 0.000, C 0.000 }
gfCNCPoint4[18732] = {X 441.4697, Y 20.1235, Z -3.6194, A 0.000, B 0.000, C 0.000 }
gfCNCPoint4[18733] = {X 441.3668, Y 20.1589, Z -3.6486, A 0.000, B 0.000, C 0.000 }
gfCNCPoint4[18734] = {X 441.1890, Y 20.7185, Z -3.8059, A 0.000, B 0.000, C 0.000 }
gfCNCPoint4[18735] = {X 441.1553, Y 21.8879, Z -4.1194, A 0.000, B 0.000, C 0.000 }
gfCNCPoint4[18736] = {X 441.2736, Y 22.3513, Z -4.2475, A 0.000, B 0.000, C 0.000 }
gfCNCPoint4[18737] = {X 441.5034, Y 22.4264, Z -4.3123, A 0.000, B 0.000, C 0.000 }
gfCNCPoint4[18738] = {X 441.7441, Y 22.4482, Z -4.3771, A 0.000, B 0.000, C 0.000 }
gfCNCPoint4[18739] = {X 443.0039, Y 22.5625, Z -4.7160, A 0.000, B 0.000, C 0.000 }
gfCNCPoint4[18740] = {X 443.1257, Y 22.5674, Z -4.7487, A 0.000, B 0.000, C 0.000 }
gfCNCPoint4[18741] = {X 444.3942, Y 22.5560, Z -5.0886, A 0.000, B 0.000, C 0.000 }
gfCNCPoint4[18742] = {X 445.9296, Y 22.5560, Z -5.5000, A 0.000, B 0.000, C 0.000 }
gfCNCPoint4[18743] = {X 450.1184, Y 22.5560, Z -5.5000, A 0.000, B 0.000, C 0.000 }
gfCNCPoint4[18744] = {X 450.1184, Y 19.7822, Z -5.5000, A 0.000, B 0.000, C 0.000 }
gfCNCPoint4[18745] = {X 444.0414, Y 19.7821, Z -5.5000, A 0.000, B 0.000, C 0.000 }
gfCNCPoint4[18746] = {X 443.3487, Y 19.7983, Z -5.5000, A 0.000, B 0.000, C 0.000 }
gfCNCPoint4[18747] = {X 442.3962, Y 19.8855, Z -5.5000, A 0.000, B 0.000, C 0.000 }
gfCNCPoint4[18748] = {X 441.4697, Y 20.1235, Z -5.5000, A 0.000, B 0.000, C 0.000 }
gfCNCPoint4[18749] = {X 441.3853, Y 20.1770, Z -5.5000, A 0.000, B 0.000, C 0.000 }
gfCNCPoint4[18750] = {X 441.3338, Y 20.2627, Z -5.5000, A 0.000, B 0.000, C 0.000 }
gfCNCPoint4[18751] = {X 441.1837, Y 20.9511, Z -5.5000, A 0.000, B 0.000, C 0.000 }
gfCNCPoint4[18752] = {X 441.1635, Y 21.6554, Z -5.5000, A 0.000, B 0.000, C 0.000 }
gfCNCPoint4[18753] = {X 441.2736, Y 22.3513, Z -5.5000, A 0.000, B 0.000, C 0.000 }
gfCNCPoint4[18754] = {X 441.5061, Y 22.4130, Z -5.5000, A 0.000, B 0.000, C 0.000 }
gfCNCPoint4[18755] = {X 441.7441, Y 22.4482, Z -5.5000, A 0.000, B 0.000, C 0.000 }
gfCNCPoint4[18756] = {X 443.0678, Y 22.5351, Z -5.5000, A 0.000, B 0.000, C 0.000 }
gfCNCPoint4[18757] = {X 444.3942, Y 22.5560, Z -5.5000, A 0.000, B 0.000, C 0.000 }
gfCNCPoint4[18758] = {X 445.9296, Y 22.5560, Z -5.5000, A 0.000, B 0.000, C 0.000 }
gfCNCPoint4[18759] = {X 441.9448, Y 22.2874, Z -5.5000, A 0.000, B 0.000, C 0.000 }
gfCNCPoint4[18760] = {X 445.9296, Y 22.6360, Z -5.5000, A 0.000, B 0.000, C 0.000 }
gfCNCPoint4[18761] = {X 450.1984, Y 22.6360, Z -5.5000, A 0.000, B 0.000, C 0.000 }
gfCNCPoint4[18762] = {X 450.1984, Y 19.7022, Z -5.5000, A 0.000, B 0.000, C 0.000 }
gfCNCPoint4[18763] = {X 444.0404, Y 19.7021, Z -5.5000, A 0.000, B 0.000, C 0.000 }
gfCNCPoint4[18764] = {X 443.3497, Y 19.7183, Z -5.5000, A 0.000, B 0.000, C 0.000 }
gfCNCPoint4[18765] = {X 442.3835, Y 19.8065, Z -5.5000, A 0.000, B 0.000, C 0.000 }
gfCNCPoint4[18766] = {X 441.4437, Y 20.0479, Z -5.5000, A 0.000, B 0.000, C 0.000 }
gfCNCPoint4[18767] = {X 441.3280, Y 20.1211, Z -5.5000, A 0.000, B 0.000, C 0.000 }
gfCNCPoint4[18768] = {X 441.2576, Y 20.2385, Z -5.5000, A 0.000, B 0.000, C 0.000 }
gfCNCPoint4[18769] = {X 441.1026, Y 20.9558, Z -5.5000, A 0.000, B 0.000, C 0.000 }
gfCNCPoint4[18770] = {X 441.0856, Y 21.6895, Z -5.5000, A 0.000, B 0.000, C 0.000 }
gfCNCPoint4[18771] = {X 441.2071, Y 22.4132, Z -5.5000, A 0.000, B 0.000, C 0.000 }
gfCNCPoint4[18772] = {X 441.4685, Y 22.4868, Z -5.5000, A 0.000, B 0.000, C 0.000 }
gfCNCPoint4[18773] = {X 441.7368, Y 22.5279, Z -5.5000, A 0.000, B 0.000, C 0.000 }
gfCNCPoint4[18774] = {X 443.0635, Y 22.6150, Z -5.5000, A 0.000, B 0.000, C 0.000 }
gfCNCPoint4[18775] = {X 444.3928, Y 22.6360, Z -5.5000, A 0.000, B 0.000, C 0.000 }
gfCNCPoint4[18776] = {X 445.9296, Y 22.6360, Z -5.5000, A 0.000, B 0.000, C 0.000 }
gfCNCPoint4[18777] = {X 449.9144, Y 22.2874, Z -5.5000, A 0.000, B 0.000, C 0.000 }
gfCNCPoint4[18778] = {X 441.9448, Y 22.3674, Z -5.5000, A 0.000, B 0.000, C 0.000 }
gfCNCPoint4[18779] = {X 445.9296, Y 22.7160, Z -5.5000, A 0.000, B 0.000, C 0.000 }
gfCNCPoint4[18780] = {X 450.2784, Y 22.7160, Z -5.5000, A 0.000, B 0.000, C 0.000 }
gfCNCPoint4[18781] = {X 450.2784, Y 19.6222, Z -5.5000, A 0.000, B 0.000, C 0.000 }
gfCNCPoint4[18782] = {X 444.0395, Y 19.6221, Z -5.5000, A 0.000, B 0.000, C 0.000 }
gfCNCPoint4[18783] = {X 443.3483, Y 19.6383, Z -5.5000, A 0.000, B 0.000, C 0.000 }
gfCNCPoint4[18784] = {X 442.3696, Y 19.7278, Z -5.5000, A 0.000, B 0.000, C 0.000 }
gfCNCPoint4[18785] = {X 441.4177, Y 19.9722, Z -5.5000, A 0.000, B 0.000, C 0.000 }
gfCNCPoint4[18786] = {X 441.2708, Y 20.0652, Z -5.5000, A 0.000, B 0.000, C 0.000 }
gfCNCPoint4[18787] = {X 441.1813, Y 20.2143, Z -5.5000, A 0.000, B 0.000, C 0.000 }
gfCNCPoint4[18788] = {X 441.0215, Y 20.9603, Z -5.5000, A 0.000, B 0.000, C 0.000 }
gfCNCPoint4[18789] = {X 441.0079, Y 21.7232, Z -5.5000, A 0.000, B 0.000, C 0.000 }
gfCNCPoint4[18790] = {X 441.1409, Y 22.4744, Z -5.5000, A 0.000, B 0.000, C 0.000 }
gfCNCPoint4[18791] = {X 441.4309, Y 22.5604, Z -5.5000, A 0.000, B 0.000, C 0.000 }
gfCNCPoint4[18792] = {X 441.7296, Y 22.6076, Z -5.5000, A 0.000, B 0.000, C 0.000 }
gfCNCPoint4[18793] = {X 443.0600, Y 22.6949, Z -5.5000, A 0.000, B 0.000, C 0.000 }
gfCNCPoint4[18794] = {X 444.3932, Y 22.7160, Z -5.5000, A 0.000, B 0.000, C 0.000 }
gfCNCPoint4[18795] = {X 445.9296, Y 22.7160, Z -5.5000, A 0.000, B 0.000, C 0.000 }
gfCNCPoint4[18796] = {X 449.9144, Y 22.3674, Z -5.5000, A 0.000, B 0.000, C 0.000 }
gfCNCPoint4[18797] = {X 441.9448, Y 22.4474, Z -5.5000, A 0.000, B 0.000, C 0.000 }
gfCNCPoint4[18798] = {X 445.9296, Y 22.7960, Z -5.5000, A 0.000, B 0.000, C 0.000 }
gfCNCPoint4[18799] = {X 450.3584, Y 22.7960, Z -5.5000, A 0.000, B 0.000, C 0.000 }
gfCNCPoint4[18800] = {X 450.3584, Y 19.5422, Z -5.5000, A 0.000, B 0.000, C 0.000 }
gfCNCPoint4[18801] = {X 444.0385, Y 19.5421, Z -5.5000, A 0.000, B 0.000, C 0.000 }
gfCNCPoint4[18802] = {X 443.3470, Y 19.5583, Z -5.5000, A 0.000, B 0.000, C 0.000 }
gfCNCPoint4[18803] = {X 442.3557, Y 19.6490, Z -5.5000, A 0.000, B 0.000, C 0.000 }
gfCNCPoint4[18804] = {X 441.3916, Y 19.8966, Z -5.5000, A 0.000, B 0.000, C 0.000 }
gfCNCPoint4[18805] = {X 441.2135, Y 20.0093, Z -5.5000, A 0.000, B 0.000, C 0.000 }
gfCNCPoint4[18806] = {X 441.1051, Y 20.1901, Z -5.5000, A 0.000, B 0.000, C 0.000 }
gfCNCPoint4[18807] = {X 440.9405, Y 20.9646, Z -5.5000, A 0.000, B 0.000, C 0.000 }
gfCNCPoint4[18808] = {X 440.9304, Y 21.7564, Z -5.5000, A 0.000, B 0.000, C 0.000 }
gfCNCPoint4[18809] = {X 441.0750, Y 22.5349, Z -5.5000, A 0.000, B 0.000, C 0.000 }
gfCNCPoint4[18810] = {X 441.3933, Y 22.6339, Z -5.5000, A 0.000, B 0.000, C 0.000 }
gfCNCPoint4[18811] = {X 441.7224, Y 22.6872, Z -5.5000, A 0.000, B 0.000, C 0.000 }
gfCNCPoint4[18812] = {X 443.0566, Y 22.7748, Z -5.5000, A 0.000, B 0.000, C 0.000 }
gfCNCPoint4[18813] = {X 444.3935, Y 22.7960, Z -5.5000, A 0.000, B 0.000, C 0.000 }
gfCNCPoint4[18814] = {X 445.9296, Y 22.7960, Z -5.5000, A 0.000, B 0.000, C 0.000 }
gfCNCPoint4[18815] = {X 449.9144, Y 22.4474, Z -5.5000, A 0.000, B 0.000, C 0.000 }
gfCNCPoint4[18816] = {X 441.9448, Y 22.5274, Z -5.5000, A 0.000, B 0.000, C 0.000 }
gfCNCPoint4[18817] = {X 445.9296, Y 22.8760, Z -5.5000, A 0.000, B 0.000, C 0.000 }
gfCNCPoint4[18818] = {X 450.4384, Y 22.8760, Z -5.5000, A 0.000, B 0.000, C 0.000 }
gfCNCPoint4[18819] = {X 450.4384, Y 19.4622, Z -5.5000, A 0.000, B 0.000, C 0.000 }
gfCNCPoint4[18820] = {X 444.0376, Y 19.4621, Z -5.5000, A 0.000, B 0.000, C 0.000 }
gfCNCPoint4[18821] = {X 443.3456, Y 19.4783, Z -5.5000, A 0.000, B 0.000, C 0.000 }
gfCNCPoint4[18822] = {X 442.3418, Y 19.5702, Z -5.5000, A 0.000, B 0.000, C 0.000 }
gfCNCPoint4[18823] = {X 441.3656, Y 19.8209, Z -5.5000, A 0.000, B 0.000, C 0.000 }
gfCNCPoint4[18824] = {X 441.1563, Y 19.9534, Z -5.5000, A 0.000, B 0.000, C 0.000 }
gfCNCPoint4[18825] = {X 441.0288, Y 20.1659, Z -5.5000, A 0.000, B 0.000, C 0.000 }
gfCNCPoint4[18826] = {X 440.8596, Y 20.9688, Z -5.5000, A 0.000, B 0.000, C 0.000 }
gfCNCPoint4[18827] = {X 440.8530, Y 21.7893, Z -5.5000, A 0.000, B 0.000, C 0.000 }
gfCNCPoint4[18828] = {X 441.0092, Y 22.5948, Z -5.5000, A 0.000, B 0.000, C 0.000 }
gfCNCPoint4[18829] = {X 441.3558, Y 22.7072, Z -5.5000, A 0.000, B 0.000, C 0.000 }
gfCNCPoint4[18830] = {X 441.7151, Y 22.7669, Z -5.5000, A 0.000, B 0.000, C 0.000 }
gfCNCPoint4[18831] = {X 443.0532, Y 22.8548, Z -5.5000, A 0.000, B 0.000, C 0.000 }
gfCNCPoint4[18832] = {X 444.3939, Y 22.8760, Z -5.5000, A 0.000, B 0.000, C 0.000 }
gfCNCPoint4[18833] = {X 445.9296, Y 22.8760, Z -5.5000, A 0.000, B 0.000, C 0.000 }
gfCNCPoint4[18834] = {X 449.9144, Y 22.5274, Z -5.5000, A 0.000, B 0.000, C 0.000 }
gfCNCPoint4[18835] = {X 445.9296, Y 20.9560, Z -5.5000, A 0.000, B 0.000, C 0.000 }
gfCNCPoint4[18836] = {X 445.9296, Y 22.9560, Z -5.5000, A 0.000, B 0.000, C 0.000 }
gfCNCPoint4[18837] = {X 450.5184, Y 22.9560, Z -5.5000, A 0.000, B 0.000, C 0.000 }
gfCNCPoint4[18838] = {X 450.5187, Y 19.3822, Z -5.5000, A 0.000, B 0.000, C 0.000 }
gfCNCPoint4[18839] = {X 444.0367, Y 19.3821, Z -5.5000, A 0.000, B 0.000, C 0.000 }
gfCNCPoint4[18840] = {X 443.3442, Y 19.3983, Z -5.5000, A 0.000, B 0.000, C 0.000 }
gfCNCPoint4[18841] = {X 442.3279, Y 19.4914, Z -5.5000, A 0.000, B 0.000, C 0.000 }
gfCNCPoint4[18842] = {X 441.3396, Y 19.7453, Z -5.5000, A 0.000, B 0.000, C 0.000 }
gfCNCPoint4[18843] = {X 441.0990, Y 19.8976, Z -5.5000, A 0.000, B 0.000, C 0.000 }
gfCNCPoint4[18844] = {X 440.9526, Y 20.1416, Z -5.5000, A 0.000, B 0.000, C 0.000 }
gfCNCPoint4[18845] = {X 440.7787, Y 20.9728, Z -5.5000, A 0.000, B 0.000, C 0.000 }
gfCNCPoint4[18846] = {X 440.7757, Y 21.8219, Z -5.5000, A 0.000, B 0.000, C 0.000 }
gfCNCPoint4[18847] = {X 440.9437, Y 22.6542, Z -5.5000, A 0.000, B 0.000, C 0.000 }
gfCNCPoint4[18848] = {X 441.3183, Y 22.7803, Z -5.5000, A 0.000, B 0.000, C 0.000 }
gfCNCPoint4[18849] = {X 441.7079, Y 22.8466, Z -5.5000, A 0.000, B 0.000, C 0.000 }
gfCNCPoint4[18850] = {X 443.0497, Y 22.9347, Z -5.5000, A 0.000, B 0.000, C 0.000 }
gfCNCPoint4[18851] = {X 444.3942, Y 22.9560, Z -5.5000, A 0.000, B 0.000, C 0.000 }
gfCNCPoint4[18852] = {X 445.9296, Y 22.9560, Z -5.5000, A 0.000, B 0.000, C 0.000 }
gfCNCPoint4[18853] = {X 449.9296, Y 22.9560, Z -5.5000, A 0.000, B 0.000, C 0.000 }
gfCNCPoint4[18854] = {X 449.9296, Y 22.9560, Z -2.5000, A 0.000, B 0.000, C 0.000 }
gfCNCPoint4[18855] = {X 449.9296, Y 22.9560, Z 11.0000, A 0.000, B 0.000, C 0.000 }
gfCNCPoint4[18856] = {X 491.9920, Y 19.7819, Z 11.0000, A 0.000, B 0.000, C 0.000 }
gfCNCPoint4[18857] = {X 491.9920, Y 19.7819, Z -1.6667, A 0.000, B 0.000, C 0.000 }
gfCNCPoint4[18858] = {X 487.6645, Y 19.7814, Z -2.8262, A 0.000, B 0.000, C 0.000 }
gfCNCPoint4[18859] = {X 486.9696, Y 19.7861, Z -3.0124, A 0.000, B 0.000, C 0.000 }
gfCNCPoint4[18860] = {X 486.2691, Y 19.7843, Z -3.2001, A 0.000, B 0.000, C 0.000 }
gfCNCPoint4[18861] = {X 485.4743, Y 19.8898, Z -3.4150, A 0.000, B 0.000, C 0.000 }
gfCNCPoint4[18862] = {X 484.7985, Y 20.0742, Z -3.6027, A 0.000, B 0.000, C 0.000 }
gfCNCPoint4[18863] = {X 484.6641, Y 20.1109, Z -3.6400, A 0.000, B 0.000, C 0.000 }
gfCNCPoint4[18864] = {X 484.6318, Y 20.1413, Z -3.6519, A 0.000, B 0.000, C 0.000 }
gfCNCPoint4[18865] = {X 484.4394, Y 20.7129, Z -3.8135, A 0.000, B 0.000, C 0.000 }
gfCNCPoint4[18866] = {X 484.4047, Y 21.9067, Z -4.1335, A 0.000, B 0.000, C 0.000 }
gfCNCPoint4[18867] = {X 484.5270, Y 22.3541, Z -4.2578, A 0.000, B 0.000, C 0.000 }
gfCNCPoint4[18868] = {X 484.7220, Y 22.4175, Z -4.3127, A 0.000, B 0.000, C 0.000 }
gfCNCPoint4[18869] = {X 484.9348, Y 22.4352, Z -4.3699, A 0.000, B 0.000, C 0.000 }
gfCNCPoint4[18870] = {X 486.0989, Y 22.5567, Z -4.6835, A 0.000, B 0.000, C 0.000 }
gfCNCPoint4[18871] = {X 486.4687, Y 22.5733, Z -4.7827, A 0.000, B 0.000, C 0.000 }
gfCNCPoint4[18872] = {X 487.6448, Y 22.5560, Z -5.0979, A 0.000, B 0.000, C 0.000 }
gfCNCPoint4[18873] = {X 489.1455, Y 22.5560, Z -5.5000, A 0.000, B 0.000, C 0.000 }
gfCNCPoint4[18874] = {X 493.3690, Y 22.5560, Z -5.5000, A 0.000, B 0.000, C 0.000 }
gfCNCPoint4[18875] = {X 493.3690, Y 19.7821, Z -5.5000, A 0.000, B 0.000, C 0.000 }
gfCNCPoint4[18876] = {X 487.6645, Y 19.7814, Z -5.5000, A 0.000, B 0.000, C 0.000 }
gfCNCPoint4[18877] = {X 486.9696, Y 19.7861, Z -5.5000, A 0.000, B 0.000, C 0.000 }
gfCNCPoint4[18878] = {X 485.8743, Y 19.8570, Z -5.5000, A 0.000, B 0.000, C 0.000 }
gfCNCPoint4[18879] = {X 484.7985, Y 20.0742, Z -5.5000, A 0.000, B 0.000, C 0.000 }
gfCNCPoint4[18880] = {X 484.6681, Y 20.1474, Z -5.5000, A 0.000, B 0.000, C 0.000 }
gfCNCPoint4[18881] = {X 484.5874, Y 20.2733, Z -5.5000, A 0.000, B 0.000, C 0.000 }
gfCNCPoint4[18882] = {X 484.4297, Y 20.9584, Z -5.5000, A 0.000, B 0.000, C 0.000 }
gfCNCPoint4[18883] = {X 484.4094, Y 21.6611, Z -5.5000, A 0.000, B 0.000, C 0.000 }
gfCNCPoint4[18884] = {X 484.5270, Y 22.3541, Z -5.5000, A 0.000, B 0.000, C 0.000 }
gfCNCPoint4[18885] = {X 484.7285, Y 22.4067, Z -5.5000, A 0.000, B 0.000, C 0.000 }
gfCNCPoint4[18886] = {X 484.9348, Y 22.4352, Z -5.5000, A 0.000, B 0.000, C 0.000 }
gfCNCPoint4[18887] = {X 486.2880, Y 22.5359, Z -5.5000, A 0.000, B 0.000, C 0.000 }
gfCNCPoint4[18888] = {X 487.6448, Y 22.5560, Z -5.5000, A 0.000, B 0.000, C 0.000 }
gfCNCPoint4[18889] = {X 489.1455, Y 22.5560, Z -5.5000, A 0.000, B 0.000, C 0.000 }
gfCNCPoint4[18890] = {X 485.1607, Y 22.2874, Z -5.5000, A 0.000, B 0.000, C 0.000 }
gfCNCPoint4[18891] = {X 489.1455, Y 22.6360, Z -5.5000, A 0.000, B 0.000, C 0.000 }
gfCNCPoint4[18892] = {X 493.4490, Y 22.6360, Z -5.5000, A 0.000, B 0.000, C 0.000 }
gfCNCPoint4[18893] = {X 493.4490, Y 19.7021, Z -5.5000, A 0.000, B 0.000, C 0.000 }
gfCNCPoint4[18894] = {X 487.6642, Y 19.7014, Z -5.5000, A 0.000, B 0.000, C 0.000 }
gfCNCPoint4[18895] = {X 486.9713, Y 19.7062, Z -5.5000, A 0.000, B 0.000, C 0.000 }
gfCNCPoint4[18896] = {X 485.8646, Y 19.7776, Z -5.5000, A 0.000, B 0.000, C 0.000 }
gfCNCPoint4[18897] = {X 484.7774, Y 19.9970, Z -5.5000, A 0.000, B 0.000, C 0.000 }
gfCNCPoint4[18898] = {X 484.6132, Y 20.0892, Z -5.5000, A 0.000, B 0.000, C 0.000 }
gfCNCPoint4[18899] = {X 484.5116, Y 20.2478, Z -5.5000, A 0.000, B 0.000, C 0.000 }
gfCNCPoint4[18900] = {X 484.3486, Y 20.9623, Z -5.5000, A 0.000, B 0.000, C 0.000 }
gfCNCPoint4[18901] = {X 484.3316, Y 21.6950, Z -5.5000, A 0.000, B 0.000, C 0.000 }
gfCNCPoint4[18902] = {X 484.4613, Y 22.4164, Z -5.5000, A 0.000, B 0.000, C 0.000 }
gfCNCPoint4[18903] = {X 484.6886, Y 22.4801, Z -5.5000, A 0.000, B 0.000, C 0.000 }
gfCNCPoint4[18904] = {X 484.9221, Y 22.5143, Z -5.5000, A 0.000, B 0.000, C 0.000 }
gfCNCPoint4[18905] = {X 486.2805, Y 22.6157, Z -5.5000, A 0.000, B 0.000, C 0.000 }
gfCNCPoint4[18906] = {X 487.6424, Y 22.6360, Z -5.5000, A 0.000, B 0.000, C 0.000 }
gfCNCPoint4[18907] = {X 489.1455, Y 22.6360, Z -5.5000, A 0.000, B 0.000, C 0.000 }
gfCNCPoint4[18908] = {X 493.1302, Y 22.2874, Z -5.5000, A 0.000, B 0.000, C 0.000 }
gfCNCPoint4[18909] = {X 485.1607, Y 22.3674, Z -5.5000, A 0.000, B 0.000, C 0.000 }
gfCNCPoint4[18910] = {X 489.1455, Y 22.7160, Z -5.5000, A 0.000, B 0.000, C 0.000 }
gfCNCPoint4[18911] = {X 493.5290, Y 22.7160, Z -5.5000, A 0.000, B 0.000, C 0.000 }
gfCNCPoint4[18912] = {X 493.5290, Y 19.6221, Z -5.5000, A 0.000, B 0.000, C 0.000 }
gfCNCPoint4[18913] = {X 487.6640, Y 19.6214, Z -5.5000, A 0.000, B 0.000, C 0.000 }
gfCNCPoint4[18914] = {X 486.9712, Y 19.6262, Z -5.5000, A 0.000, B 0.000, C 0.000 }
gfCNCPoint4[18915] = {X 485.8539, Y 19.6984, Z -5.5000, A 0.000, B 0.000, C 0.000 }
gfCNCPoint4[18916] = {X 484.7564, Y 19.9198, Z -5.5000, A 0.000, B 0.000, C 0.000 }
gfCNCPoint4[18917] = {X 484.5583, Y 20.0310, Z -5.5000, A 0.000, B 0.000, C 0.000 }
gfCNCPoint4[18918] = {X 484.4358, Y 20.2223, Z -5.5000, A 0.000, B 0.000, C 0.000 }
gfCNCPoint4[18919] = {X 484.2676, Y 20.9660, Z -5.5000, A 0.000, B 0.000, C 0.000 }
gfCNCPoint4[18920] = {X 484.2541, Y 21.7285, Z -5.5000, A 0.000, B 0.000, C 0.000 }
gfCNCPoint4[18921] = {X 484.3959, Y 22.4777, Z -5.5000, A 0.000, B 0.000, C 0.000 }
gfCNCPoint4[18922] = {X 484.6513, Y 22.5539, Z -5.5000, A 0.000, B 0.000, C 0.000 }
gfCNCPoint4[18923] = {X 484.9147, Y 22.5940, Z -5.5000, A 0.000, B 0.000, C 0.000 }
gfCNCPoint4[18924] = {X 486.2770, Y 22.6956, Z -5.5000, A 0.000, B 0.000, C 0.000 }
gfCNCPoint4[18925] = {X 487.6430, Y 22.7160, Z -5.5000, A 0.000, B 0.000, C 0.000 }
gfCNCPoint4[18926] = {X 489.1455, Y 22.7160, Z -5.5000, A 0.000, B 0.000, C 0.000 }
gfCNCPoint4[18927] = {X 493.1302, Y 22.3674, Z -5.5000, A 0.000, B 0.000, C 0.000 }
gfCNCPoint4[18928] = {X 485.1607, Y 22.4474, Z -5.5000, A 0.000, B 0.000, C 0.000 }
gfCNCPoint4[18929] = {X 489.1455, Y 22.7960, Z -5.5000, A 0.000, B 0.000, C 0.000 }
gfCNCPoint4[18930] = {X 493.6090, Y 22.7960, Z -5.5000, A 0.000, B 0.000, C 0.000 }
gfCNCPoint4[18931] = {X 493.6090, Y 19.5421, Z -5.5000, A 0.000, B 0.000, C 0.000 }
gfCNCPoint4[18932] = {X 487.6637, Y 19.5414, Z -5.5000, A 0.000, B 0.000, C 0.000 }
gfCNCPoint4[18933] = {X 486.9710, Y 19.5462, Z -5.5000, A 0.000, B 0.000, C 0.000 }
gfCNCPoint4[18934] = {X 485.8432, Y 19.6191, Z -5.5000, A 0.000, B 0.000, C 0.000 }
gfCNCPoint4[18935] = {X 484.7353, Y 19.8427, Z -5.5000, A 0.000, B 0.000, C 0.000 }
gfCNCPoint4[18936] = {X 484.5034, Y 19.9728, Z -5.5000, A 0.000, B 0.000, C 0.000 }
gfCNCPoint4[18937] = {X 484.3599, Y 20.1968, Z -5.5000, A 0.000, B 0.000, C 0.000 }
gfCNCPoint4[18938] = {X 484.1866, Y 20.9695, Z -5.5000, A 0.000, B 0.000, C 0.000 }
gfCNCPoint4[18939] = {X 484.1767, Y 21.7614, Z -5.5000, A 0.000, B 0.000, C 0.000 }
gfCNCPoint4[18940] = {X 484.3307, Y 22.5382, Z -5.5000, A 0.000, B 0.000, C 0.000 }
gfCNCPoint4[18941] = {X 484.6139, Y 22.6274, Z -5.5000, A 0.000, B 0.000, C 0.000 }
gfCNCPoint4[18942] = {X 484.9072, Y 22.6736, Z -5.5000, A 0.000, B 0.000, C 0.000 }
gfCNCPoint4[18943] = {X 486.2736, Y 22.7755, Z -5.5000, A 0.000, B 0.000, C 0.000 }
gfCNCPoint4[18944] = {X 487.6436, Y 22.7960, Z -5.5000, A 0.000, B 0.000, C 0.000 }
gfCNCPoint4[18945] = {X 489.1455, Y 22.7960, Z -5.5000, A 0.000, B 0.000, C 0.000 }
gfCNCPoint4[18946] = {X 493.1302, Y 22.4474, Z -5.5000, A 0.000, B 0.000, C 0.000 }
gfCNCPoint4[18947] = {X 485.1607, Y 22.5274, Z -5.5000, A 0.000, B 0.000, C 0.000 }
gfCNCPoint4[18948] = {X 489.1455, Y 22.8760, Z -5.5000, A 0.000, B 0.000, C 0.000 }
gfCNCPoint4[18949] = {X 493.6890, Y 22.8760, Z -5.5000, A 0.000, B 0.000, C 0.000 }
gfCNCPoint4[18950] = {X 493.6890, Y 19.4621, Z -5.5000, A 0.000, B 0.000, C 0.000 }
gfCNCPoint4[18951] = {X 487.6634, Y 19.4614, Z -5.5000, A 0.000, B 0.000, C 0.000 }
gfCNCPoint4[18952] = {X 486.9708, Y 19.4661, Z -5.5000, A 0.000, B 0.000, C 0.000 }
gfCNCPoint4[18953] = {X 485.8325, Y 19.5398, Z -5.5000, A 0.000, B 0.000, C 0.000 }
gfCNCPoint4[18954] = {X 484.7142, Y 19.7655, Z -5.5000, A 0.000, B 0.000, C 0.000 }
gfCNCPoint4[18955] = {X 484.4485, Y 19.9146, Z -5.5000, A 0.000, B 0.000, C 0.000 }
gfCNCPoint4[18956] = {X 484.2841, Y 20.1712, Z -5.5000, A 0.000, B 0.000, C 0.000 }
gfCNCPoint4[18957] = {X 484.1057, Y 20.9728, Z -5.5000, A 0.000, B 0.000, C 0.000 }
gfCNCPoint4[18958] = {X 484.0994, Y 21.7939, Z -5.5000, A 0.000, B 0.000, C 0.000 }
gfCNCPoint4[18959] = {X 484.2656, Y 22.5981, Z -5.5000, A 0.000, B 0.000, C 0.000 }
gfCNCPoint4[18960] = {X 484.5770, Y 22.7008, Z -5.5000, A 0.000, B 0.000, C 0.000 }
gfCNCPoint4[18961] = {X 484.9007, Y 22.7534, Z -5.5000, A 0.000, B 0.000, C 0.000 }
gfCNCPoint4[18962] = {X 486.2706, Y 22.8555, Z -5.5000, A 0.000, B 0.000, C 0.000 }
gfCNCPoint4[18963] = {X 487.6442, Y 22.8760, Z -5.5000, A 0.000, B 0.000, C 0.000 }
gfCNCPoint4[18964] = {X 489.1455, Y 22.8760, Z -5.5000, A 0.000, B 0.000, C 0.000 }
gfCNCPoint4[18965] = {X 493.1302, Y 22.5274, Z -5.5000, A 0.000, B 0.000, C 0.000 }
gfCNCPoint4[18966] = {X 489.1455, Y 20.9560, Z -5.5000, A 0.000, B 0.000, C 0.000 }
gfCNCPoint4[18967] = {X 489.1455, Y 22.9560, Z -5.5000, A 0.000, B 0.000, C 0.000 }
gfCNCPoint4[18968] = {X 493.7690, Y 22.9560, Z -5.5000, A 0.000, B 0.000, C 0.000 }
gfCNCPoint4[18969] = {X 493.7693, Y 19.3821, Z -5.5000, A 0.000, B 0.000, C 0.000 }
gfCNCPoint4[18970] = {X 487.6632, Y 19.3814, Z -5.5000, A 0.000, B 0.000, C 0.000 }
gfCNCPoint4[18971] = {X 486.9707, Y 19.3861, Z -5.5000, A 0.000, B 0.000, C 0.000 }
gfCNCPoint4[18972] = {X 485.8217, Y 19.4605, Z -5.5000, A 0.000, B 0.000, C 0.000 }
gfCNCPoint4[18973] = {X 484.6932, Y 19.6883, Z -5.5000, A 0.000, B 0.000, C 0.000 }
gfCNCPoint4[18974] = {X 484.3936, Y 19.8564, Z -5.5000, A 0.000, B 0.000, C 0.000 }
gfCNCPoint4[18975] = {X 484.2083, Y 20.1457, Z -5.5000, A 0.000, B 0.000, C 0.000 }
gfCNCPoint4[18976] = {X 484.0248, Y 20.9758, Z -5.5000, A 0.000, B 0.000, C 0.000 }
gfCNCPoint4[18977] = {X 484.0223, Y 21.8260, Z -5.5000, A 0.000, B 0.000, C 0.000 }
gfCNCPoint4[18978] = {X 484.2007, Y 22.6572, Z -5.5000, A 0.000, B 0.000, C 0.000 }
gfCNCPoint4[18979] = {X 484.5397, Y 22.7739, Z -5.5000, A 0.000, B 0.000, C 0.000 }
gfCNCPoint4[18980] = {X 484.8932, Y 22.8330, Z -5.5000, A 0.000, B 0.000, C 0.000 }
gfCNCPoint4[18981] = {X 486.2672, Y 22.9354, Z -5.5000, A 0.000, B 0.000, C 0.000 }
gfCNCPoint4[18982] = {X 487.6448, Y 22.9560, Z -5.5000, A 0.000, B 0.000, C 0.000 }
gfCNCPoint4[18983] = {X 489.1455, Y 22.9560, Z -5.5000, A 0.000, B 0.000, C 0.000 }
gfCNCPoint4[18984] = {X 493.1455, Y 22.9560, Z -5.5000, A 0.000, B 0.000, C 0.000 }
gfCNCPoint4[18985] = {X 493.1455, Y 22.9560, Z -2.5000, A 0.000, B 0.000, C 0.000 }
gfCNCPoint4[18986] = {X 493.1455, Y 22.9560, Z 11.0000, A 0.000, B 0.000, C 0.000 }
gfCNCPoint4[18987] = {X 607.6966, Y 2.1245, Z 11.0000, A 0.000, B 0.000, C 0.000 }
gfCNCPoint4[18988] = {X 607.6966, Y 2.1245, Z -2.5000, A 0.000, B 0.000, C 0.000 }
gfCNCPoint4[18989] = {X 607.6966, Y 2.1245, Z -5.5000, A 0.000, B 0.000, C 0.000 }
gfCNCPoint4[18990] = {X 603.6966, Y 8.3205, Z -5.5000, A 0.000, B 0.000, C 0.000 }
gfCNCPoint4[18991] = {X 603.3207, Y 8.8207, Z -5.5000, A 0.000, B 0.000, C 0.000 }
gfCNCPoint4[18992] = {X 602.8777, Y 9.2625, Z -5.5000, A 0.000, B 0.000, C 0.000 }
gfCNCPoint4[18993] = {X 602.8775, Y 40.7373, Z -5.5000, A 0.000, B 0.000, C 0.000 }
gfCNCPoint4[18994] = {X 603.3207, Y 41.1792, Z -5.5000, A 0.000, B 0.000, C 0.000 }
gfCNCPoint4[18995] = {X 603.6966, Y 41.6795, Z -5.5000, A 0.000, B 0.000, C 0.000 }
gfCNCPoint4[18996] = {X 607.6966, Y 47.8755, Z -5.5000, A 0.000, B 0.000, C 0.000 }
gfCNCPoint4[18997] = {X 607.6966, Y 47.8755, Z -2.5000, A 0.000, B 0.000, C 0.000 }
gfCNCPoint4[18998] = {X 607.6966, Y 47.8755, Z 11.0000, A 0.000, B 0.000, C 0.000 }
gfCNCPoint4[18999] = {X 607.6966, Y 1.5466, Z 11.0000, A 0.000, B 0.000, C 0.000 }
gfCNCPoint4[19000] = {X 607.6966, Y 1.5466, Z -2.5000, A 0.000, B 0.000, C 0.000 }
gfCNCPoint4[19001] = {X 607.6966, Y 1.5466, Z -5.5000, A 0.000, B 0.000, C 0.000 }
gfCNCPoint4[19002] = {X 603.6966, Y 8.1707, Z -5.5000, A 0.000, B 0.000, C 0.000 }
gfCNCPoint4[19003] = {X 603.2899, Y 8.7357, Z -5.5000, A 0.000, B 0.000, C 0.000 }
gfCNCPoint4[19004] = {X 602.7977, Y 9.2280, Z -5.5000, A 0.000, B 0.000, C 0.000 }
gfCNCPoint4[19005] = {X 602.7975, Y 40.7725, Z -5.5000, A 0.000, B 0.000, C 0.000 }
gfCNCPoint4[19006] = {X 603.2898, Y 41.2648, Z -5.5000, A 0.000, B 0.000, C 0.000 }
gfCNCPoint4[19007] = {X 603.6966, Y 41.8297, Z -5.5000, A 0.000, B 0.000, C 0.000 }
gfCNCPoint4[19008] = {X 607.6966, Y 48.4506, Z -5.5000, A 0.000, B 0.000, C 0.000 }
gfCNCPoint4[19009] = {X 607.6966, Y 48.4506, Z -2.5000, A 0.000, B 0.000, C 0.000 }
gfCNCPoint4[19010] = {X 607.6966, Y 48.4506, Z 11.0000, A 0.000, B 0.000, C 0.000 }
gfCNCPoint4[19011] = {X 607.6966, Y 0.8798, Z 11.0000, A 0.000, B 0.000, C 0.000 }
gfCNCPoint4[19012] = {X 607.6966, Y 0.8798, Z -2.5000, A 0.000, B 0.000, C 0.000 }
gfCNCPoint4[19013] = {X 607.6966, Y 0.8798, Z -5.5000, A 0.000, B 0.000, C 0.000 }
gfCNCPoint4[19014] = {X 603.6966, Y 8.0117, Z -5.5000, A 0.000, B 0.000, C 0.000 }
gfCNCPoint4[19015] = {X 603.2609, Y 8.6459, Z -5.5000, A 0.000, B 0.000, C 0.000 }
gfCNCPoint4[19016] = {X 602.7177, Y 9.1909, Z -5.5000, A 0.000, B 0.000, C 0.000 }
gfCNCPoint4[19017] = {X 602.7175, Y 40.8097, Z -5.5000, A 0.000, B 0.000, C 0.000 }
gfCNCPoint4[19018] = {X 603.2608, Y 41.3546, Z -5.5000, A 0.000, B 0.000, C 0.000 }
gfCNCPoint4[19019] = {X 603.6966, Y 41.9886, Z -5.5000, A 0.000, B 0.000, C 0.000 }
gfCNCPoint4[19020] = {X 607.6966, Y 49.1167, Z -5.5000, A 0.000, B 0.000, C 0.000 }
gfCNCPoint4[19021] = {X 607.6966, Y 49.1167, Z -2.5000, A 0.000, B 0.000, C 0.000 }
gfCNCPoint4[19022] = {X 607.6966, Y 49.1167, Z 11.0000, A 0.000, B 0.000, C 0.000 }
gfCNCPoint4[19023] = {X 607.6951, Y 0.0817, Z 11.0000, A 0.000, B 0.000, C 0.000 }
gfCNCPoint4[19024] = {X 607.6951, Y 0.0817, Z -2.5000, A 0.000, B 0.000, C 0.000 }
gfCNCPoint4[19025] = {X 607.6951, Y 0.0817, Z -5.5000, A 0.000, B 0.000, C 0.000 }
gfCNCPoint4[19026] = {X 603.6966, Y 7.8428, Z -5.5000, A 0.000, B 0.000, C 0.000 }
gfCNCPoint4[19027] = {X 603.2342, Y 8.5522, Z -5.5000, A 0.000, B 0.000, C 0.000 }
gfCNCPoint4[19028] = {X 602.6377, Y 9.1532, Z -5.5000, A 0.000, B 0.000, C 0.000 }
gfCNCPoint4[19029] = {X 602.6375, Y 40.8474, Z -5.5000, A 0.000, B 0.000, C 0.000 }
gfCNCPoint4[19030] = {X 603.2341, Y 41.4482, Z -5.5000, A 0.000, B 0.000, C 0.000 }
gfCNCPoint4[19031] = {X 603.6966, Y 42.1574, Z -5.5000, A 0.000, B 0.000, C 0.000 }
gfCNCPoint4[19032] = {X 607.6966, Y 49.9167, Z -5.5000, A 0.000, B 0.000, C 0.000 }
gfCNCPoint4[19033] = {X 607.6966, Y 49.9167, Z -2.5000, A 0.000, B 0.000, C 0.000 }
gfCNCPoint4[19034] = {X 607.6966, Y 49.9167, Z 11.0000, A 0.000, B 0.000, C 0.000 }
gfCNCPoint4[19035] = {X 607.6538, Y -0.8109, Z 11.0000, A 0.000, B 0.000, C 0.000 }
gfCNCPoint4[19036] = {X 607.6538, Y -0.8109, Z -2.5000, A 0.000, B 0.000, C 0.000 }
gfCNCPoint4[19037] = {X 607.6538, Y -0.8109, Z -5.5000, A 0.000, B 0.000, C 0.000 }
gfCNCPoint4[19038] = {X 603.6966, Y 7.6608, Z -5.5000, A 0.000, B 0.000, C 0.000 }
gfCNCPoint4[19039] = {X 603.2073, Y 8.4559, Z -5.5000, A 0.000, B 0.000, C 0.000 }
gfCNCPoint4[19040] = {X 602.5500, Y 9.1190, Z -5.5000, A 0.000, B 0.000, C 0.000 }
gfCNCPoint4[19041] = {X 602.5577, Y 9.1532, Z -5.5000, A 0.000, B 0.000, C 0.000 }
gfCNCPoint4[19042] = {X 602.5575, Y 40.8854, Z -5.5000, A 0.000, B 0.000, C 0.000 }
gfCNCPoint4[19043] = {X 603.2104, Y 41.5469, Z -5.5000, A 0.000, B 0.000, C 0.000 }
gfCNCPoint4[19044] = {X 603.6966, Y 42.3390, Z -5.5000, A 0.000, B 0.000, C 0.000 }
gfCNCPoint4[19045] = {X 607.6966, Y 50.9152, Z -5.5000, A 0.000, B 0.000, C 0.000 }
gfCNCPoint4[19046] = {X 607.6966, Y 50.9152, Z -2.5000, A 0.000, B 0.000, C 0.000 }
gfCNCPoint4[19047] = {X 607.6966, Y 50.9152, Z 11.0000, A 0.000, B 0.000, C 0.000 }
gfCNCPoint4[19048] = {X 607.4986, Y -1.7352, Z 11.0000, A 0.000, B 0.000, C 0.000 }
gfCNCPoint4[19049] = {X 607.4986, Y -1.7352, Z -2.5000, A 0.000, B 0.000, C 0.000 }
gfCNCPoint4[19050] = {X 607.4986, Y -1.7352, Z -5.5000, A 0.000, B 0.000, C 0.000 }
gfCNCPoint4[19051] = {X 603.6966, Y 7.4622, Z -5.5000, A 0.000, B 0.000, C 0.000 }
gfCNCPoint4[19052] = {X 603.3769, Y 8.0780, Z -5.5000, A 0.000, B 0.000, C 0.000 }
gfCNCPoint4[19053] = {X 602.9556, Y 8.6293, Z -5.5000, A 0.000, B 0.000, C 0.000 }
gfCNCPoint4[19054] = {X 602.4454, Y 9.0995, Z -5.5000, A 0.000, B 0.000, C 0.000 }
gfCNCPoint4[19055] = {X 602.4777, Y 9.1532, Z -5.5000, A 0.000, B 0.000, C 0.000 }
gfCNCPoint4[19056] = {X 602.4775, Y 40.9225, Z -5.5000, A 0.000, B 0.000, C 0.000 }
gfCNCPoint4[19057] = {X 602.5729, Y 41.0032, Z -5.5000, A 0.000, B 0.000, C 0.000 }
gfCNCPoint4[19058] = {X 603.2273, Y 41.7028, Z -5.5000, A 0.000, B 0.000, C 0.000 }
gfCNCPoint4[19059] = {X 603.6966, Y 42.5378, Z -5.5000, A 0.000, B 0.000, C 0.000 }
gfCNCPoint4[19060] = {X 607.6966, Y 52.2141, Z -5.5000, A 0.000, B 0.000, C 0.000 }
gfCNCPoint4[19061] = {X 607.6966, Y 52.2141, Z -2.5000, A 0.000, B 0.000, C 0.000 }
gfCNCPoint4[19062] = {X 607.6966, Y 52.2141, Z 11.0000, A 0.000, B 0.000, C 0.000 }
gfCNCPoint4[19063] = {X 607.6966, Y 2.1243, Z 11.0000, A 0.000, B 0.000, C 0.000 }
gfCNCPoint4[19064] = {X 607.6966, Y 2.1243, Z -3.3333, A 0.000, B 0.000, C 0.000 }
gfCNCPoint4[19065] = {X 607.6966, Y 2.1243, Z -6.3333, A 0.000, B 0.000, C 0.000 }
gfCNCPoint4[19066] = {X 603.6966, Y 8.3205, Z -6.3333, A 0.000, B 0.000, C 0.000 }
gfCNCPoint4[19067] = {X 603.3209, Y 8.8205, Z -6.3333, A 0.000, B 0.000, C 0.000 }
gfCNCPoint4[19068] = {X 602.8780, Y 9.2623, Z -6.3333, A 0.000, B 0.000, C 0.000 }
gfCNCPoint4[19069] = {X 602.8778, Y 40.7376, Z -6.3333, A 0.000, B 0.000, C 0.000 }
gfCNCPoint4[19070] = {X 603.3208, Y 41.1794, Z -6.3333, A 0.000, B 0.000, C 0.000 }
gfCNCPoint4[19071] = {X 603.6966, Y 41.6795, Z -6.3333, A 0.000, B 0.000, C 0.000 }
gfCNCPoint4[19072] = {X 607.6966, Y 47.8757, Z -6.3333, A 0.000, B 0.000, C 0.000 }
gfCNCPoint4[19073] = {X 607.6966, Y 47.8757, Z -3.3333, A 0.000, B 0.000, C 0.000 }
gfCNCPoint4[19074] = {X 607.6966, Y 47.8757, Z 11.0000, A 0.000, B 0.000, C 0.000 }
gfCNCPoint4[19075] = {X 607.6966, Y 1.5453, Z 11.0000, A 0.000, B 0.000, C 0.000 }
gfCNCPoint4[19076] = {X 607.6966, Y 1.5453, Z -3.3333, A 0.000, B 0.000, C 0.000 }
gfCNCPoint4[19077] = {X 607.6966, Y 1.5453, Z -6.3333, A 0.000, B 0.000, C 0.000 }
gfCNCPoint4[19078] = {X 603.6966, Y 8.1708, Z -6.3333, A 0.000, B 0.000, C 0.000 }
gfCNCPoint4[19079] = {X 603.2901, Y 8.7357, Z -6.3333, A 0.000, B 0.000, C 0.000 }
gfCNCPoint4[19080] = {X 602.7980, Y 9.2280, Z -6.3333, A 0.000, B 0.000, C 0.000 }
gfCNCPoint4[19081] = {X 602.7978, Y 40.7725, Z -6.3333, A 0.000, B 0.000, C 0.000 }
gfCNCPoint4[19082] = {X 603.2900, Y 41.2647, Z -6.3333, A 0.000, B 0.000, C 0.000 }
gfCNCPoint4[19083] = {X 603.6966, Y 41.8296, Z -6.3333, A 0.000, B 0.000, C 0.000 }
gfCNCPoint4[19084] = {X 607.6966, Y 48.4519, Z -6.3333, A 0.000, B 0.000, C 0.000 }
gfCNCPoint4[19085] = {X 607.6966, Y 48.4519, Z -3.3333, A 0.000, B 0.000, C 0.000 }
gfCNCPoint4[19086] = {X 607.6966, Y 48.4519, Z 11.0000, A 0.000, B 0.000, C 0.000 }
gfCNCPoint4[19087] = {X 607.6966, Y 0.8783, Z 11.0000, A 0.000, B 0.000, C 0.000 }
gfCNCPoint4[19088] = {X 607.6966, Y 0.8783, Z -3.3333, A 0.000, B 0.000, C 0.000 }
gfCNCPoint4[19089] = {X 607.6966, Y 0.8783, Z -6.3333, A 0.000, B 0.000, C 0.000 }
gfCNCPoint4[19090] = {X 603.6966, Y 8.0118, Z -6.3333, A 0.000, B 0.000, C 0.000 }
gfCNCPoint4[19091] = {X 603.2610, Y 8.6459, Z -6.3333, A 0.000, B 0.000, C 0.000 }
gfCNCPoint4[19092] = {X 602.7180, Y 9.1909, Z -6.3333, A 0.000, B 0.000, C 0.000 }
gfCNCPoint4[19093] = {X 602.7178, Y 40.8097, Z -6.3333, A 0.000, B 0.000, C 0.000 }
gfCNCPoint4[19094] = {X 603.2609, Y 41.3546, Z -6.3333, A 0.000, B 0.000, C 0.000 }
gfCNCPoint4[19095] = {X 603.6966, Y 41.9885, Z -6.3333, A 0.000, B 0.000, C 0.000 }
gfCNCPoint4[19096] = {X 607.6966, Y 49.1182, Z -6.3333, A 0.000, B 0.000, C 0.000 }
gfCNCPoint4[19097] = {X 607.6966, Y 49.1182, Z -3.3333, A 0.000, B 0.000, C 0.000 }
gfCNCPoint4[19098] = {X 607.6966, Y 49.1182, Z 11.0000, A 0.000, B 0.000, C 0.000 }
gfCNCPoint4[19099] = {X 607.6951, Y 0.0798, Z 11.0000, A 0.000, B 0.000, C 0.000 }
gfCNCPoint4[19100] = {X 607.6951, Y 0.0798, Z -3.3333, A 0.000, B 0.000, C 0.000 }
gfCNCPoint4[19101] = {X 607.6951, Y 0.0798, Z -6.3333, A 0.000, B 0.000, C 0.000 }
gfCNCPoint4[19102] = {X 603.6966, Y 7.8429, Z -6.3333, A 0.000, B 0.000, C 0.000 }
gfCNCPoint4[19103] = {X 603.2344, Y 8.5522, Z -6.3333, A 0.000, B 0.000, C 0.000 }
gfCNCPoint4[19104] = {X 602.6380, Y 9.1532, Z -6.3333, A 0.000, B 0.000, C 0.000 }
gfCNCPoint4[19105] = {X 602.6378, Y 40.8473, Z -6.3333, A 0.000, B 0.000, C 0.000 }
gfCNCPoint4[19106] = {X 603.2342, Y 41.4482, Z -6.3333, A 0.000, B 0.000, C 0.000 }
gfCNCPoint4[19107] = {X 603.6966, Y 42.1574, Z -6.3333, A 0.000, B 0.000, C 0.000 }
gfCNCPoint4[19108] = {X 607.6966, Y 49.9187, Z -6.3333, A 0.000, B 0.000, C 0.000 }
gfCNCPoint4[19109] = {X 607.6966, Y 49.9187, Z -3.3333, A 0.000, B 0.000, C 0.000 }
gfCNCPoint4[19110] = {X 607.6966, Y 49.9187, Z 11.0000, A 0.000, B 0.000, C 0.000 }
gfCNCPoint4[19111] = {X 607.6538, Y -0.8113, Z 11.0000, A 0.000, B 0.000, C 0.000 }
gfCNCPoint4[19112] = {X 607.6538, Y -0.8113, Z -3.3333, A 0.000, B 0.000, C 0.000 }
gfCNCPoint4[19113] = {X 607.6538, Y -0.8113, Z -6.3333, A 0.000, B 0.000, C 0.000 }
gfCNCPoint4[19114] = {X 603.6966, Y 7.6607, Z -6.3333, A 0.000, B 0.000, C 0.000 }
gfCNCPoint4[19115] = {X 603.2074, Y 8.4558, Z -6.3333, A 0.000, B 0.000, C 0.000 }
gfCNCPoint4[19116] = {X 602.5503, Y 9.1188, Z -6.3333, A 0.000, B 0.000, C 0.000 }
gfCNCPoint4[19117] = {X 602.5580, Y 9.1532, Z -6.3333, A 0.000, B 0.000, C 0.000 }
gfCNCPoint4[19118] = {X 602.5578, Y 40.8854, Z -6.3333, A 0.000, B 0.000, C 0.000 }
gfCNCPoint4[19119] = {X 603.2106, Y 41.5469, Z -6.3333, A 0.000, B 0.000, C 0.000 }
gfCNCPoint4[19120] = {X 603.6966, Y 42.3390, Z -6.3333, A 0.000, B 0.000, C 0.000 }
gfCNCPoint4[19121] = {X 607.6966, Y 50.9178, Z -6.3333, A 0.000, B 0.000, C 0.000 }
gfCNCPoint4[19122] = {X 607.6966, Y 50.9178, Z -3.3333, A 0.000, B 0.000, C 0.000 }
gfCNCPoint4[19123] = {X 607.6966, Y 50.9178, Z 11.0000, A 0.000, B 0.000, C 0.000 }
gfCNCPoint4[19124] = {X 607.4985, Y -1.7355, Z 11.0000, A 0.000, B 0.000, C 0.000 }
gfCNCPoint4[19125] = {X 607.4985, Y -1.7355, Z -3.3333, A 0.000, B 0.000, C 0.000 }
gfCNCPoint4[19126] = {X 607.4985, Y -1.7355, Z -6.3333, A 0.000, B 0.000, C 0.000 }
gfCNCPoint4[19127] = {X 603.6966, Y 7.4621, Z -6.3333, A 0.000, B 0.000, C 0.000 }
gfCNCPoint4[19128] = {X 603.3770, Y 8.0779, Z -6.3333, A 0.000, B 0.000, C 0.000 }
gfCNCPoint4[19129] = {X 602.9557, Y 8.6293, Z -6.3333, A 0.000, B 0.000, C 0.000 }
gfCNCPoint4[19130] = {X 602.4454, Y 9.0995, Z -6.3333, A 0.000, B 0.000, C 0.000 }
gfCNCPoint4[19131] = {X 602.4780, Y 9.1532, Z -6.3333, A 0.000, B 0.000, C 0.000 }
gfCNCPoint4[19132] = {X 602.4778, Y 40.9224, Z -6.3333, A 0.000, B 0.000, C 0.000 }
gfCNCPoint4[19133] = {X 602.5730, Y 41.0033, Z -6.3333, A 0.000, B 0.000, C 0.000 }
gfCNCPoint4[19134] = {X 603.2274, Y 41.7029, Z -6.3333, A 0.000, B 0.000, C 0.000 }
gfCNCPoint4[19135] = {X 603.6966, Y 42.5379, Z -6.3333, A 0.000, B 0.000, C 0.000 }
gfCNCPoint4[19136] = {X 607.6966, Y 52.2148, Z -6.3333, A 0.000, B 0.000, C 0.000 }
gfCNCPoint4[19137] = {X 607.6966, Y 52.2148, Z -3.3333, A 0.000, B 0.000, C 0.000 }
gfCNCPoint4[19138] = {X 607.6966, Y 52.2148, Z 11.0000, A 0.000, B 0.000, C 0.000 }
gfCNCPoint4[19139] = {X 491.9930, Y 19.7822, Z 11.0000, A 0.000, B 0.000, C 0.000 }
gfCNCPoint4[19140] = {X 491.9930, Y 19.7822, Z -2.5000, A 0.000, B 0.000, C 0.000 }
gfCNCPoint4[19141] = {X 487.6645, Y 19.7817, Z -3.6598, A 0.000, B 0.000, C 0.000 }
gfCNCPoint4[19142] = {X 486.9696, Y 19.7865, Z -3.8460, A 0.000, B 0.000, C 0.000 }
gfCNCPoint4[19143] = {X 486.2691, Y 19.7846, Z -4.0337, A 0.000, B 0.000, C 0.000 }
gfCNCPoint4[19144] = {X 485.4746, Y 19.8900, Z -4.2485, A 0.000, B 0.000, C 0.000 }
gfCNCPoint4[19145] = {X 484.7988, Y 20.0745, Z -4.4362, A 0.000, B 0.000, C 0.000 }
gfCNCPoint4[19146] = {X 484.6643, Y 20.1112, Z -4.4735, A 0.000, B 0.000, C 0.000 }
gfCNCPoint4[19147] = {X 484.6315, Y 20.1421, Z -4.4856, A 0.000, B 0.000, C 0.000 }
gfCNCPoint4[19148] = {X 484.5872, Y 20.2743, Z -4.5230, A 0.000, B 0.000, C 0.000 }
gfCNCPoint4[19149] = {X 484.4395, Y 20.7146, Z -4.6474, A 0.000, B 0.000, C 0.000 }
gfCNCPoint4[19150] = {X 484.4051, Y 21.9058, Z -4.9667, A 0.000, B 0.000, C 0.000 }
gfCNCPoint4[19151] = {X 484.5272, Y 22.3538, Z -5.0912, A 0.000, B 0.000, C 0.000 }
gfCNCPoint4[19152] = {X 484.7221, Y 22.4171, Z -5.1461, A 0.000, B 0.000, C 0.000 }
gfCNCPoint4[19153] = {X 484.9348, Y 22.4349, Z -5.2033, A 0.000, B 0.000, C 0.000 }
gfCNCPoint4[19154] = {X 486.1009, Y 22.5565, Z -5.5174, A 0.000, B 0.000, C 0.000 }
gfCNCPoint4[19155] = {X 486.4667, Y 22.5729, Z -5.6155, A 0.000, B 0.000, C 0.000 }
gfCNCPoint4[19156] = {X 487.6448, Y 22.5560, Z -5.9312, A 0.000, B 0.000, C 0.000 }
gfCNCPoint4[19157] = {X 489.1455, Y 22.5560, Z -6.3333, A 0.000, B 0.000, C 0.000 }
gfCNCPoint4[19158] = {X 493.3690, Y 22.5560, Z -6.3333, A 0.000, B 0.000, C 0.000 }
gfCNCPoint4[19159] = {X 493.3690, Y 19.7823, Z -6.3333, A 0.000, B 0.000, C 0.000 }
gfCNCPoint4[19160] = {X 487.6645, Y 19.7817, Z -6.3333, A 0.000, B 0.000, C 0.000 }
gfCNCPoint4[19161] = {X 486.9696, Y 19.7865, Z -6.3333, A 0.000, B 0.000, C 0.000 }
gfCNCPoint4[19162] = {X 485.8745, Y 19.8574, Z -6.3333, A 0.000, B 0.000, C 0.000 }
gfCNCPoint4[19163] = {X 484.7988, Y 20.0745, Z -6.3333, A 0.000, B 0.000, C 0.000 }
gfCNCPoint4[19164] = {X 484.6680, Y 20.1479, Z -6.3333, A 0.000, B 0.000, C 0.000 }
gfCNCPoint4[19165] = {X 484.5872, Y 20.2743, Z -6.3333, A 0.000, B 0.000, C 0.000 }
gfCNCPoint4[19166] = {X 484.4302, Y 20.9590, Z -6.3333, A 0.000, B 0.000, C 0.000 }
gfCNCPoint4[19167] = {X 484.4099, Y 21.6612, Z -6.3333, A 0.000, B 0.000, C 0.000 }
gfCNCPoint4[19168] = {X 484.5272, Y 22.3538, Z -6.3333, A 0.000, B 0.000, C 0.000 }
gfCNCPoint4[19169] = {X 484.7286, Y 22.4064, Z -6.3333, A 0.000, B 0.000, C 0.000 }
gfCNCPoint4[19170] = {X 484.9348, Y 22.4349, Z -6.3333, A 0.000, B 0.000, C 0.000 }
gfCNCPoint4[19171] = {X 486.2880, Y 22.5356, Z -6.3333, A 0.000, B 0.000, C 0.000 }
gfCNCPoint4[19172] = {X 487.6448, Y 22.5560, Z -6.3333, A 0.000, B 0.000, C 0.000 }
gfCNCPoint4[19173] = {X 489.1455, Y 22.5560, Z -6.3333, A 0.000, B 0.000, C 0.000 }
gfCNCPoint4[19174] = {X 485.1607, Y 22.2874, Z -6.3333, A 0.000, B 0.000, C 0.000 }
gfCNCPoint4[19175] = {X 489.1455, Y 22.6360, Z -6.3333, A 0.000, B 0.000, C 0.000 }
gfCNCPoint4[19176] = {X 493.4490, Y 22.6360, Z -6.3333, A 0.000, B 0.000, C 0.000 }
gfCNCPoint4[19177] = {X 493.4490, Y 19.7024, Z -6.3333, A 0.000, B 0.000, C 0.000 }
gfCNCPoint4[19178] = {X 487.6642, Y 19.7017, Z -6.3333, A 0.000, B 0.000, C 0.000 }
gfCNCPoint4[19179] = {X 486.9713, Y 19.7065, Z -6.3333, A 0.000, B 0.000, C 0.000 }
gfCNCPoint4[19180] = {X 485.8647, Y 19.7780, Z -6.3333, A 0.000, B 0.000, C 0.000 }
gfCNCPoint4[19181] = {X 484.7777, Y 19.9973, Z -6.3333, A 0.000, B 0.000, C 0.000 }
gfCNCPoint4[19182] = {X 484.6130, Y 20.0897, Z -6.3333, A 0.000, B 0.000, C 0.000 }
gfCNCPoint4[19183] = {X 484.5113, Y 20.2488, Z -6.3333, A 0.000, B 0.000, C 0.000 }
gfCNCPoint4[19184] = {X 484.3490, Y 20.9630, Z -6.3333, A 0.000, B 0.000, C 0.000 }
gfCNCPoint4[19185] = {X 484.3322, Y 21.6952, Z -6.3333, A 0.000, B 0.000, C 0.000 }
gfCNCPoint4[19186] = {X 484.4615, Y 22.4161, Z -6.3333, A 0.000, B 0.000, C 0.000 }
gfCNCPoint4[19187] = {X 484.6882, Y 22.4797, Z -6.3333, A 0.000, B 0.000, C 0.000 }
gfCNCPoint4[19188] = {X 484.9212, Y 22.5139, Z -6.3333, A 0.000, B 0.000, C 0.000 }
gfCNCPoint4[19189] = {X 486.2800, Y 22.6153, Z -6.3333, A 0.000, B 0.000, C 0.000 }
gfCNCPoint4[19190] = {X 487.6425, Y 22.6360, Z -6.3333, A 0.000, B 0.000, C 0.000 }
gfCNCPoint4[19191] = {X 489.1455, Y 22.6360, Z -6.3333, A 0.000, B 0.000, C 0.000 }
gfCNCPoint4[19192] = {X 493.1302, Y 22.2874, Z -6.3333, A 0.000, B 0.000, C 0.000 }
gfCNCPoint4[19193] = {X 485.1607, Y 22.3674, Z -6.3333, A 0.000, B 0.000, C 0.000 }
gfCNCPoint4[19194] = {X 489.1455, Y 22.7160, Z -6.3333, A 0.000, B 0.000, C 0.000 }
gfCNCPoint4[19195] = {X 493.5290, Y 22.7160, Z -6.3333, A 0.000, B 0.000, C 0.000 }
gfCNCPoint4[19196] = {X 493.5290, Y 19.6224, Z -6.3333, A 0.000, B 0.000, C 0.000 }
gfCNCPoint4[19197] = {X 487.6640, Y 19.6217, Z -6.3333, A 0.000, B 0.000, C 0.000 }
gfCNCPoint4[19198] = {X 486.9712, Y 19.6265, Z -6.3333, A 0.000, B 0.000, C 0.000 }
gfCNCPoint4[19199] = {X 485.8540, Y 19.6987, Z -6.3333, A 0.000, B 0.000, C 0.000 }
gfCNCPoint4[19200] = {X 484.7566, Y 19.9201, Z -6.3333, A 0.000, B 0.000, C 0.000 }
gfCNCPoint4[19201] = {X 484.5581, Y 20.0316, Z -6.3333, A 0.000, B 0.000, C 0.000 }
gfCNCPoint4[19202] = {X 484.4355, Y 20.2234, Z -6.3333, A 0.000, B 0.000, C 0.000 }
gfCNCPoint4[19203] = {X 484.2680, Y 20.9667, Z -6.3333, A 0.000, B 0.000, C 0.000 }
gfCNCPoint4[19204] = {X 484.2546, Y 21.7286, Z -6.3333, A 0.000, B 0.000, C 0.000 }
gfCNCPoint4[19205] = {X 484.3960, Y 22.4774, Z -6.3333, A 0.000, B 0.000, C 0.000 }
gfCNCPoint4[19206] = {X 484.6513, Y 22.5535, Z -6.3333, A 0.000, B 0.000, C 0.000 }
gfCNCPoint4[19207] = {X 484.9147, Y 22.5937, Z -6.3333, A 0.000, B 0.000, C 0.000 }
gfCNCPoint4[19208] = {X 486.2771, Y 22.6953, Z -6.3333, A 0.000, B 0.000, C 0.000 }
gfCNCPoint4[19209] = {X 487.6431, Y 22.7160, Z -6.3333, A 0.000, B 0.000, C 0.000 }
gfCNCPoint4[19210] = {X 489.1455, Y 22.7160, Z -6.3333, A 0.000, B 0.000, C 0.000 }
gfCNCPoint4[19211] = {X 493.1302, Y 22.3674, Z -6.3333, A 0.000, B 0.000, C 0.000 }
gfCNCPoint4[19212] = {X 485.1607, Y 22.4474, Z -6.3333, A 0.000, B 0.000, C 0.000 }
gfCNCPoint4[19213] = {X 489.1455, Y 22.7960, Z -6.3333, A 0.000, B 0.000, C 0.000 }
gfCNCPoint4[19214] = {X 493.6090, Y 22.7960, Z -6.3333, A 0.000, B 0.000, C 0.000 }
gfCNCPoint4[19215] = {X 493.6090, Y 19.5424, Z -6.3333, A 0.000, B 0.000, C 0.000 }
gfCNCPoint4[19216] = {X 487.6637, Y 19.5417, Z -6.3333, A 0.000, B 0.000, C 0.000 }
gfCNCPoint4[19217] = {X 486.9710, Y 19.5465, Z -6.3333, A 0.000, B 0.000, C 0.000 }
gfCNCPoint4[19218] = {X 485.8433, Y 19.6194, Z -6.3333, A 0.000, B 0.000, C 0.000 }
gfCNCPoint4[19219] = {X 484.7356, Y 19.8429, Z -6.3333, A 0.000, B 0.000, C 0.000 }
gfCNCPoint4[19220] = {X 484.5032, Y 19.9734, Z -6.3333, A 0.000, B 0.000, C 0.000 }
gfCNCPoint4[19221] = {X 484.3596, Y 20.1979, Z -6.3333, A 0.000, B 0.000, C 0.000 }
gfCNCPoint4[19222] = {X 484.1870, Y 20.9703, Z -6.3333, A 0.000, B 0.000, C 0.000 }
gfCNCPoint4[19223] = {X 484.1772, Y 21.7616, Z -6.3333, A 0.000, B 0.000, C 0.000 }
gfCNCPoint4[19224] = {X 484.3307, Y 22.5379, Z -6.3333, A 0.000, B 0.000, C 0.000 }
gfCNCPoint4[19225] = {X 484.6140, Y 22.6270, Z -6.3333, A 0.000, B 0.000, C 0.000 }
gfCNCPoint4[19226] = {X 484.9072, Y 22.6733, Z -6.3333, A 0.000, B 0.000, C 0.000 }
gfCNCPoint4[19227] = {X 486.2736, Y 22.7752, Z -6.3333, A 0.000, B 0.000, C 0.000 }
gfCNCPoint4[19228] = {X 487.6436, Y 22.7960, Z -6.3333, A 0.000, B 0.000, C 0.000 }
gfCNCPoint4[19229] = {X 489.1455, Y 22.7960, Z -6.3333, A 0.000, B 0.000, C 0.000 }
gfCNCPoint4[19230] = {X 493.1302, Y 22.4474, Z -6.3333, A 0.000, B 0.000, C 0.000 }
